(* CODESYS project Tc3_Physics.library
   TcLibraryId: Beckhoff Automation GmbH|Tc3_Physics|0.3.79.0
   Company: Beckhoff Automation GmbH
   DefaultNamespace: Tc3_Physics
   Version: 0.3.79.0
   Placeholder: Tc3_Physics
   Title: Tc3_Physics

Project tree, tasks and I/O mapping:
  Version/
    global variables Global_Version
  POUs/
    Spatial/
      Functions/
        function ConcatenateXY [ST]
        function Concatenate3D [ST]
        function ConcatenateC [ST]
        function ConcatenateABC [ST]
        function ConcatenateXYC [ST]
        function Concatenate6D [ST]
        function AddXY [ST]
        function SubtractXY [ST]
        function MultiplyXY [ST]
        function ScalarXY [ST]
        function Add3D [ST]
        function Subtract3D [ST]
        function Multiply3D [ST]
        function Scalar3D [ST]
        function Cross3D [ST]
        function AddABC [ST]
        function SubtractABC [ST]
        function MultiplyABC [ST]
        function AddXYC [ST]
        function SubtractXYC [ST]
        function MultiplyXYC [ST]
        function Add6D [ST]
        function Subtract6D [ST]
        function Multiply6D [ST]
        function ConvertToCartesian2D [ST]
      Positions/
        function block PositionXY [ST]: FB_init, FB_reinit, FB_exit, SetZero, SetValues, SetValuesXY, SetValuesRP, SetValuesXYReferenceId, GetRadius, GetPhi, Invert, ConcatenateWith, ShiftBy, ShiftByXY, x, y, ReferenceId
        function block Position3D [ST]: FB_init, FB_exit, SetZero, SetValues, SetValuesXYZ, SetValuesRPZ, SetValuesRTP, Invert, ConcatenateWith, ShiftBy, ShiftByXYZ, x, y, z
        function block Orientation2D [ST]: FB_init, FB_exit, SetAngle, SetZero, SetValues, GetDirectionX, GetDirectionY, Invert, ConcatenateWith, TurnByC, Transform, angle
        function block Orientation3D [ST]: FB_init, FB_exit, SetZero, SetValues, SetValuesABC, SetValuesACB, SetValuesBCA, SetValuesBAC, SetValuesCAB, SetValuesCBA, SetValuesABA, SetValuesACA, SetValuesBCB, SetValuesBAB, SetValuesCAC, SetValuesCBC, GetDirectionX, GetDirectionY, GetDirectionZ, Invert, ConcatenateWith, TurnBy, TurnByA, TurnByB, TurnByC, Transform, phi0, phi1, phi2, convention
        function block PositionXYC [ST]: FB_init, FB_reinit, FB_exit, SetZero, SetValues, SetValuesXY, SetValuesXYC, SetValuesXYCReferenceId, GetDirectionX, GetDirectionY, Invert, ConcatenateWith, StepByLocal, StepByLocalXY, ShiftBy, ShiftByXY, TurnByC, Transform, x, y, c, ReferenceId
        function block PositionSE3 [ST]: FB_init, FB_exit, SetZero, SetValues, SetValuesXYZ, SetValuesRPZ, SetValuesRTP, SetValuesABC, SetValuesACB, SetValuesBCA, SetValuesBAC, SetValuesCAB, SetValuesCBA, SetValuesABA, SetValuesACA, SetValuesBCB, SetValuesBAB, SetValuesCAC, SetValuesCBC, GetDirectionX, GetDirectionY, GetDirectionZ, Invert, ConcatenateWith, StepByLocal, StepByLocalXYZ, ShiftBy, ShiftByXYZ, TurnBy, TurnByA, TurnByB, TurnByC, Transform, x, y, z, phi0, phi1, phi2, Convention
      Tangents/
        function block TangentXY [ST]: FB_init, FB_exit, SetZero, SetValues, SetValuesXY, IsZero, GetLength, GetDirection, AddBy, AddByXY, SubtractBy, SubtractByXY, MultiplyBy, Normalize, x, y
        function block Tangent3D [ST]: FB_init, FB_exit, SetZero, SetValues, SetValuesXYZ, IsZero, GetLength, GetDirection, AddBy, AddByXYZ, SubtractBy, SubtractByXYZ, MultiplyBy, DivideBy, Normalize, x, y, z
        function block TangentABC [ST]: FB_init, FB_exit, SetZero, SetValues, SetValuesABC, IsZero, GetLength, AddBy, AddByABC, SubtractBy, SubtractByABC, MultiplyBy, a, b, c
        function block TangentXYC [ST]: FB_init, FB_exit, SetZero, SetValues, SetValuesXYC, IsZero, AddBy, AddByXYC, SubtractBy, SubtractByXYC, MultiplyBy, x, y, c
        function block Tangent6D [ST]: FB_init, FB_exit
      Setpoints/
        function block SetpointR1 [ST]: FB_init, FB_reinit, FB_exit, SetZero, SetValuesSVAJ, _s, v, a, j
        function block SetpointSE3 [ST]: FB_init, FB_exit, SetIdentity, SetValues, SetValuesXYZ, SetValuesCBA, GetDirectionX, GetDirectionY, GetDirectionZ, GetPosition_Cartesian, GetVelocity_Cartesian, GetAcceleration_Cartesian, GetJerk_Cartesian, ConcatenateWith, x, y, z, phi0, phi1, phi2, Convention
      Inertias/
        function block InertiaSE3 [ST]: FB_init, FB_exit, AddBy, SetValues_Point, SetValues_Sphere, SetValues_Cylinder, SetValues_Cuboid, Transform, Translate, mass, x, y, z, xx, yy, zz, xy, yz, zx
    _Internal/
      function block IPlcGeometry2D [ST]: FB_init, FB_exit
      function block IPlcGeometry3D [ST]: FB_init, FB_exit
      function block Geometry2D [ST]: FB_init, FB_exit, SetDisplacement, SetDisplacementXYC, SetDisplacementXY, SetDisplacementX, SetDisplacementY, SetDisplacementC, SetPosition, SetPositionXYC, SetPositionXY, SetPositionX, SetPositionY, SetPositionC, GetDisplacement, GetDisplacementX, GetDisplacementY, GetDisplacementC, GetLocalX, GetLocalY, GetPosition, GetPositionX, GetPositionY, GetPositionC, GetDirectionX, GetDirectionY, StepByLocal, StepByLocalXY, ShiftBy, ShiftByXY, TurnByC
      function block Geometry3D [ST]: FB_init, FB_exit, SetDisplacement, SetDisplacementXYZ, SetDisplacementX, SetDisplacementY, SetDisplacementZ, SetPosition, SetPositionXYZ, SetPositionX, SetPositionY, SetPositionZ, SetRotationABC, SetRotationACB, SetRotationBCA, SetRotationBAC, SetRotationCAB, SetRotationCBA, SetRotationABA, SetRotationACA, SetRotationBCB, SetRotationBAB, SetRotationCAC, SetRotationCBC, GetDisplacement, GetDisplacementX, GetDisplacementY, GetDisplacementZ, GetLocalX, GetLocalY, GetLocalZ, GetPosition, GetPositionX, GetPositionY, GetPositionZ, GetDirectionX, GetDirectionY, GetDirectionZ, StepByLocal, StepByLocalXYZ, ShiftBy, ShiftByXYZ, TurnBy, TurnByA, TurnByB, TurnByC, phi0, phi1, phi2, Convention
      function block IPlcPath2D [ST]: FB_init, FB_exit, CloseLoop, Clear, GetLength, IsClosedLoop, IsSelfColliding, GetArcLength_ClosestTo
      function block IPlcPath3D [ST]: FB_init, FB_exit, CloseLoop, Clear, GetLength, IsClosedLoop, IsSelfColliding, GetArcLength_ClosestTo
      function block IPlcDynamicConstraint [ST]: FB_init, FB_exit
    Shapes/
      Geometry2D/
        1D/
          function block Line2D [ST]: FB_init, FB_exit, DefineByPositions, DefineByDirection, SetDirection, GetDirection, GetPositionAt
          function block Segment2D [ST]: FB_init, FB_exit, SetStartPosition, SetStartPositionXY, SetEndPosition, SetEndPositionXY, Get_dX, Get_dY, GetLength, GetStartPosition, GetEndPosition, GetDirection, GetPositionAt
          function block Circle2D [ST]: FB_init, FB_exit, GetLength, GetPositionAt, radius
        2D/
          function block Disc2D [ST]: FB_init, FB_exit, GetArea, radius
          function block Rectangle2D [ST]: FB_init, FB_exit, SetDimensions, GetArea, width, height
        function block Container2D [ST]: FB_init, FB_exit, AddElement, RemoveElement, Clear, GetCount, GetBoundary
        function block Extrude2D [ST]: FB_init, FB_exit, ExtrudeAlong, IsValid
        Functions/
          function CheckCollision2D [ST]
          function GetDistance2D [ST]
          function GetLinkingLine2D [ST]
      Geometry3D/
        1D/
          function block Line3D [ST]: FB_init, FB_exit, DefineByPositions, DefineByDirection, SetDirection, GetDirection, GetPositionAt
          function block Segment3D [ST]: FB_init, FB_exit, SetStartPosition, SetStartPositionXYZ, SetEndPosition, SetEndPositionXYZ, Get_dX, Get_dY, Get_dZ, GetLength, GetStartPosition, GetEndPosition, GetDirection, GetPositionAt
          function block Circle3D [ST]: FB_init, FB_exit, SetNormal, GetLength, GetNormal, GetPositionAt, radius
        2D/
          function block Plane3D [ST]: FB_init, FB_exit, SetNormal, GetNormal
          function block Disc3D [ST]: FB_init, FB_exit, SetNormal, GetNormal, GetArea, radius
          function block Rectangle3D [ST]: FB_init, FB_exit, SetDimensions, GetArea, width, height
        3D/
          function block Sphere3D [ST]: FB_init, FB_exit, GetVolume, radius
          function block Cuboid3D [ST]: FB_init, FB_exit, SetDimensions, GetVolume, length, width, height
          function block Cylinder3D [ST]: FB_init, FB_exit, SetDimensions, GetVolume, radius, height
        function block Container3D [ST]: FB_init, FB_exit, AddElement, RemoveElement, Clear, GetCount
        function block Extrude3D [ST]: FB_init, FB_exit, DefineByPath
        Functions/
          function CheckCollision3D [ST]
          function GetDistance3D [ST]
          function GetLinkingLine3D [ST]
          function CreateIntersection2D [ST]
    Paths/
      Components/
        function block PathXY [ST]: FB_init, FB_exit, AppendPosition, AppendPositionXY, AppendLine, AppendCircle, GetStartPosition, GetEndPosition, GetPositionAt, GetStateAt
        function block PathXYC [ST]: FB_init, FB_exit, AppendPosition, AppendPositionXYC, AppendLine, AppendCircle, EndAtPath, StartFromPath, CloseLoop, Clear, GetStartPosition, GetEndPosition, GetPositionAt, GetStateAt
        function block PathXYZ [ST]: FB_init, FB_exit, AppendPosition, AppendPositionXYZ, AppendLine, AppendLineXYZ, AppendCircle, AppendPositionTangent, GetStartPosition, GetEndPosition, GetPositionAt, GetStateAt
    Dynamics/
      function block DynamicConstraint_Container [ST]: FB_init, FB_exit, Clear, AddConstraint, AddConstraintByReference, Count
      function block DynamicConstraint_CartesianXY [ST]: FB_init, FB_exit, SetValuesVAJ, V, A, J
      function block DynamicConstraint_CartesianXYZ [ST]: FB_init, FB_exit, SetValuesVAJ, V, A, J
      function block DynamicConstraint_Path [ST]: FB_init, FB_exit
      function block DynamicConstraint_PathXY [ST]: FB_init, FB_exit, SetValuesVADJ, V, A, D, J
      function block DynamicConstraint_PathXYZ [ST]: FB_init, FB_exit, SetValuesVADJ, V, A, D, J
      function block DynamicConstraint_Coordinates [ST]: FB_init, FB_exit, AddLimit, SetLimit, RemoveLimit, Clear, GetV, GetA, GetD, GetJ, Count
      function block DynamicProfile_7phase [ST]: FB_init, FB_exit, SetDynamicLimits, CalculateProfile, GetValues, GetDuration
      function block DynamicProfile_3phase [ST]: FB_init, FB_exit, SetDynamicLimits, CalculateProfile, GetValues, GetDuration
    Coordinates/
      function GetMcsCoordinateType [ST]
      function GetUninterpretedCoordinateType [ST]
  DUTs/
    Enumerations/
      data type E_RotationCoordinates
      data type E_CoordCategory
      data type E_McsCoordType
    data type CoordinateType
  GVLs/
    global variables GVL
*)

// DUTs/CoordinateType

(* Coordinate type. Use provided constants such as Coord_Mcs_X or factory functions such as GetMcsCoordinateType for creation. *)
	{attribute 'TcIecLibraryType'}
TYPE CoordinateType : 
	STRUCT
		(* Reserved. *)
		{attribute 'hide'}
		_reserved0 : ULINT := 0;
	END_STRUCT
END_TYPE

// DUTs/Enumerations/E_RotationCoordinates

(* Enumeration of rotation conventions. 
			    The order of letters defines the order of rotation around local axes.
			    This also defines order in which user should program rotation values. *)
	{attribute 'TcIecLibraryType'}
{attribute 'qualified_only'}
{attribute 'strict'}
TYPE E_RotationCoordinates : (
	ABC:=0, 	(* ABC *)
	ACB:=1, 	(* ACB *)
	BCA:=2, 	(* BCA *)
	BAC:=3, 	(* BAC *)
	CAB:=4, 	(* CAB *)
	CBA:=5, 	(* CBA *)
	ABA:=6, 	(* ABA *)
	ACA:=7, 	(* ACA *)
	BCB:=8, 	(* BCB *)
	BAB:=9, 	(* BAB *)
	CAC:=10, 	(* CAC *)
	CBC:=11	(* CBC *)
) UDINT;
END_TYPE

// DUTs/Enumerations/E_CoordCategory

(* Enumeration coordinate categories. *)
	{attribute 'TcIecLibraryType'}
{attribute 'qualified_only'}
{attribute 'strict'}
TYPE E_CoordCategory : (
	Invalid:=16#0, 	(* Invalid *)
	MCS:=16#1, 	(* MCS *)
	ACS:=16#2, 	(* ACS *)
	Uninterpreted:=16#3	(* Uninterpreted *)
) UDINT;
END_TYPE

// DUTs/Enumerations/E_McsCoordType

(* Enumeration of MCS coordinate types. *)
	{attribute 'TcIecLibraryType'}
{attribute 'qualified_only'}
{attribute 'strict'}
TYPE E_McsCoordType : (
	Invalid:=16#0, 	(* Invalid *)
	X:=16#11, 	(* X *)
	Y:=16#21, 	(* Y *)
	Z:=16#31, 	(* Z *)
	A1:=16#41, 	(* A1 *)
	A2:=16#42, 	(* A2 *)
	A3:=16#43, 	(* A3 *)
	B1:=16#51, 	(* B1 *)
	B2:=16#52, 	(* B2 *)
	B3:=16#53, 	(* B3 *)
	C1:=16#61, 	(* C1 *)
	C2:=16#62, 	(* C2 *)
	C3:=16#63	(* C3 *)
) UDINT;
END_TYPE

// Version/Global_Version
{attribute 'TcGenerated'}
// This function has been automatically generated from the project information.
VAR_GLOBAL CONSTANT
	{attribute 'const_non_replaced'}
	{attribute 'linkalways'}
	stLibVersion_Tc3_Physics : ST_LibVersion := (iMajor := 0, iMinor := 3, iBuild := 79, iRevision := 0, sVersion := '0.3.79.0');
	{attribute 'const_non_replaced'}
	{attribute 'linkalways'}
	sLibraryId_Tc3_Physics : String := 'Beckhoff Automation GmbH|Tc3_Physics|0.3.79.0';
END_VAR

// GVLs/GVL

VAR_GLOBAL CONSTANT
		Coord_Mcs_X	:	CoordinateType := GetMcsCoordinateType(E_McsCoordType.X);
		Coord_Mcs_Y	:	CoordinateType := GetMcsCoordinateType(E_McsCoordType.Y);
		Coord_Mcs_Z	:	CoordinateType := GetMcsCoordinateType(E_McsCoordType.Z);
		Coord_Mcs_A1	:	CoordinateType := GetMcsCoordinateType(E_McsCoordType.A1);
		Coord_Mcs_A2	:	CoordinateType := GetMcsCoordinateType(E_McsCoordType.A2);
		Coord_Mcs_A3	:	CoordinateType := GetMcsCoordinateType(E_McsCoordType.A3);
		Coord_Mcs_B1	:	CoordinateType := GetMcsCoordinateType(E_McsCoordType.B1);
		Coord_Mcs_B2	:	CoordinateType := GetMcsCoordinateType(E_McsCoordType.B2);
		Coord_Mcs_B3	:	CoordinateType := GetMcsCoordinateType(E_McsCoordType.B3);
		Coord_Mcs_C1	:	CoordinateType := GetMcsCoordinateType(E_McsCoordType.C1);
		Coord_Mcs_C2	:	CoordinateType := GetMcsCoordinateType(E_McsCoordType.C2);
		Coord_Mcs_C3	:	CoordinateType := GetMcsCoordinateType(E_McsCoordType.C3);
		Coord_Uninterpreted1	:	CoordinateType := GetUninterpretedCoordinateType(1);
		Coord_Uninterpreted2	:	CoordinateType := GetUninterpretedCoordinateType(2);
		Coord_Uninterpreted3	:	CoordinateType := GetUninterpretedCoordinateType(3);
		Coord_Uninterpreted4	:	CoordinateType := GetUninterpretedCoordinateType(4);
		Coord_Uninterpreted5	:	CoordinateType := GetUninterpretedCoordinateType(5);
		Coord_Uninterpreted6	:	CoordinateType := GetUninterpretedCoordinateType(6);
		Coord_Uninterpreted7	:	CoordinateType := GetUninterpretedCoordinateType(7);
		Coord_Uninterpreted8	:	CoordinateType := GetUninterpretedCoordinateType(8);
	END_VAR

// POUs/_Internal/IPlcGeometry2D

	{attribute 'c++_compatible'}
	{attribute 'external_name' := 'IPlcGeometry2D_GUID_0554E5C0_4687_0E31_67FE_D976C958432A'}
	{attribute 'TcIecLibraryType'}
	{attribute 'no_explicit_call' :='do not call this POU directly'}
	{attribute 'no_assign_warning'}
	(* Internal representation of an object in the planar space. *)
	FUNCTION_BLOCK IPlcGeometry2D
	VAR
		(* x-coordinate of the instance. *)
		px : LREAL;
		(* y-coordinate of the instance. *)
		py : LREAL;
		(* c-rotation of the instance given in degrees [Â°]. *)
		pc : LREAL;
		 {attribute 'hide'}
		_reserved1 : ARRAY [1..24] OF USINT;
	END_VAR
	VAR_OUTPUT
		(* ErrorCode for last method execution *)
		nErrorId : UDINT;
		(* Error during last method execution *)
		bError : BOOL;
	END_VAR
	VAR
		 {attribute 'hide'}
		_reserved2 : ARRAY [1..35] OF USINT;
	END_VAR


	(* Internal method *)
	{attribute 'hide'}
	METHOD FB_init : BOOL
	VAR_INPUT
		(*  if TRUE, the retain variables are initialized (warm start / cold start) *)
		bInitRetains : BOOL;
		(*  if TRUE, the instance afterwards gets moved into the copy code (online change) *)
		bInCopyCode : BOOL;
	END_VAR
END_METHOD


	(* Internal method *)
	{attribute 'hide'}
	METHOD FB_exit : BOOL
	VAR_INPUT
		(*  if TRUE, the exit method is called for exiting an instance that is copied afterwards (online change). *)
		bInCopyCode : BOOL;
	END_VAR
END_METHOD

END_FUNCTION_BLOCK

// POUs/_Internal/IPlcGeometry3D

	{attribute 'c++_compatible'}
	{attribute 'external_name' := 'IPlcGeometry3D_GUID_353920C5_B103_0C39_7785_16CAA850CA31'}
	{attribute 'TcIecLibraryType'}
	{attribute 'no_explicit_call' :='do not call this POU directly'}
	{attribute 'no_assign'}
	(* Internal representation of an object in the 3D space. *)
	FUNCTION_BLOCK IPlcGeometry3D
	VAR
		(* x-coordinate of the instance. *)
		px : LREAL;
		(* y-coordinate of the instance. *)
		py : LREAL;
		(* z-coordinate of the instance. *)
		pz : LREAL;
		 {attribute 'hide'}
		_reserved1 : ARRAY [1..40] OF USINT;
	END_VAR
	VAR_OUTPUT
		(* ErrorCode for last method execution *)
		nErrorId : UDINT;
		(* Error during last method execution *)
		bError : BOOL;
	END_VAR
	VAR
		 {attribute 'hide'}
		_reserved2 : ARRAY [1..43] OF USINT;
	END_VAR


	(* Internal method *)
	{attribute 'hide'}
	METHOD FB_init : BOOL
	VAR_INPUT
		(*  if TRUE, the retain variables are initialized (warm start / cold start) *)
		bInitRetains : BOOL;
		(*  if TRUE, the instance afterwards gets moved into the copy code (online change) *)
		bInCopyCode : BOOL;
	END_VAR
END_METHOD


	(* Internal method *)
	{attribute 'hide'}
	METHOD FB_exit : BOOL
	VAR_INPUT
		(*  if TRUE, the exit method is called for exiting an instance that is copied afterwards (online change). *)
		bInCopyCode : BOOL;
	END_VAR
END_METHOD

END_FUNCTION_BLOCK

// POUs/_Internal/Geometry2D

	{attribute 'c++_compatible'}
	{attribute 'external_name' := 'Geometry2D_GUID_EA1925AE_2507_0F27_40AC_5A565B8F6BBE'}
	{attribute 'TcIecLibraryType'}
	{attribute 'no_explicit_call' :='do not call this POU directly'}
	{attribute 'no_assign'}
	(* Base class for all 2D simple geometries (all dimensions, line etc.) *)
	FUNCTION_BLOCK Geometry2D EXTENDS IPlcGeometry2D


	(* Internal method *)
	METHOD FB_init : BOOL
	VAR_INPUT
		(*  if TRUE, the retain variables are initialized (warm start / cold start) *)
		bInitRetains : BOOL;
		(*  if TRUE, the instance afterwards gets moved into the copy code (online change) *)
		bInCopyCode : BOOL;
	END_VAR
END_METHOD


	(* Internal method *)
	{attribute 'hide'}
	METHOD FB_exit : BOOL
	VAR_INPUT
		(*  if TRUE, the exit method is called for exiting an instance that is copied afterwards (online change). *)
		bInCopyCode : BOOL;
	END_VAR
END_METHOD


	(* Set the position of this geometry in respect to the reference frame. *)
	METHOD SetDisplacement
	VAR_IN_OUT
		(* The displacement to set. *)
 {attribute 'GUID' := '54EDED35-5A53-0913-4680-EA5D332AAA4F'}
				displacement : PositionXYC;
	END_VAR
END_METHOD


	(* Set the position of this geometry in respect to the reference frame. *)
	METHOD SetDisplacementXYC
	VAR_INPUT
		(* x-component of the position. *)
		x : LREAL;
		(* y-component of the position. *)
		y : LREAL;
		(* c-component of the position given in degrees [Â°]. *)
		c : LREAL;
	END_VAR
END_METHOD


	(* Set the position of this geometry in respect to the reference frame. *)
	METHOD SetDisplacementXY
	VAR_INPUT
		(* x-component of the position. *)
		x : LREAL;
		(* y-component of the position. *)
		y : LREAL;
	END_VAR
END_METHOD


	(* Set the local x-coordinate of this geometry. *)
	METHOD SetDisplacementX
	VAR_INPUT
		(* Global x-component of the position. *)
		x : LREAL;
	END_VAR
END_METHOD


	(* Set the local y-coordinate of this geometry. *)
	METHOD SetDisplacementY
	VAR_INPUT
		(* Global y-component of the position. *)
		y : LREAL;
	END_VAR
END_METHOD


	(* Set the local c-component of this geometry. *)
	METHOD SetDisplacementC
	VAR_INPUT
		(* c-orientation given in degrees [Â°]. *)
		c : LREAL;
	END_VAR
END_METHOD


	(* Set the position of this geometry in respect to the WCS. *)
	METHOD SetPosition
	VAR_IN_OUT
		(* The position to set. *)
 {attribute 'GUID' := '54EDED35-5A53-0913-4680-EA5D332AAA4F'}
				position : PositionXYC;
	END_VAR
END_METHOD


	(* Set the position of this geometry in respect to the WCS. *)
	METHOD SetPositionXYC
	VAR_INPUT
		(* x-component of the position. *)
		x : LREAL;
		(* y-component of the position. *)
		y : LREAL;
		(* c-component of the position given in degrees [Â°]. *)
		c : LREAL;
	END_VAR
END_METHOD


	(* Set the position of this geometry in respect to the WCS. *)
	METHOD SetPositionXY
	VAR_INPUT
		(* x-component of the position. *)
		x : LREAL;
		(* y-component of the position. *)
		y : LREAL;
	END_VAR
END_METHOD


	(* Set the global x-coordinate of this geometry. *)
	METHOD SetPositionX
	VAR_INPUT
		(* Global x-component of the position. *)
		x : LREAL;
	END_VAR
END_METHOD


	(* Set the global y-coordinate of this geometry. *)
	METHOD SetPositionY
	VAR_INPUT
		(* Global y-component of the position. *)
		y : LREAL;
	END_VAR
END_METHOD


	(* Set the global c-component of this geometry. *)
	METHOD SetPositionC
	VAR_INPUT
		(* c-orientation given in degrees [Â°]. *)
		c : LREAL;
	END_VAR
END_METHOD


	(* Get the position of this geometry in respect to the reference frame. *)
	METHOD GetDisplacement
	VAR_IN_OUT
		(* The current position of the geometry. *)
 {attribute 'GUID' := '54EDED35-5A53-0913-4680-EA5D332AAA4F'}
				displacement : PositionXYC;
	END_VAR
END_METHOD


	(* Get the local x-component of this geometry. *)
	METHOD GetDisplacementX : LREAL
END_METHOD


	(* Get the local y-component of this geometry. *)
	METHOD GetDisplacementY : LREAL
END_METHOD


	(* Get the local c-orientation of this geometry. *)
	METHOD GetDisplacementC : LREAL
END_METHOD


	(* Get the direction of the local x-axis. *)
	METHOD GetLocalX
	VAR_IN_OUT
		(* The local x-direction of this geometry. *)
 {attribute 'GUID' := '619D5D7D-53EC-0B73-54D5-FB9C43AFDE82'}
				localX : TangentXY;
	END_VAR
END_METHOD


	(* Get the direction of the local y-axis. *)
	METHOD GetLocalY
	VAR_IN_OUT
		(* The local y-direction of this geometry. *)
 {attribute 'GUID' := '619D5D7D-53EC-0B73-54D5-FB9C43AFDE82'}
				localY : TangentXY;
	END_VAR
END_METHOD


	(* Get the position of this geometry. *)
	METHOD GetPosition
	VAR_IN_OUT
		(* The current position of the geometry. *)
 {attribute 'GUID' := '54EDED35-5A53-0913-4680-EA5D332AAA4F'}
				position : PositionXYC;
	END_VAR
END_METHOD


	(* Get the global x-component of this geometry. *)
	METHOD GetPositionX : LREAL
END_METHOD


	(* Get the global y-component of this geometry. *)
	METHOD GetPositionY : LREAL
END_METHOD


	(* Get the global c-orientation of this geometry. *)
	METHOD GetPositionC : LREAL
END_METHOD


	(* Get the direction of the local x-axis. *)
	METHOD GetDirectionX
	VAR_IN_OUT
		(* The global x-direction of this geometry. *)
 {attribute 'GUID' := '619D5D7D-53EC-0B73-54D5-FB9C43AFDE82'}
				directionX : TangentXY;
	END_VAR
END_METHOD


	(* Get the direction of the local y-axis. *)
	METHOD GetDirectionY
	VAR_IN_OUT
		(* The global y-direction of this geometry. *)
 {attribute 'GUID' := '619D5D7D-53EC-0B73-54D5-FB9C43AFDE82'}
				directionY : TangentXY;
	END_VAR
END_METHOD


	(* Displace the components of this position. The shift is applied within the local coordinate frame. *)
	METHOD StepByLocal
	VAR_IN_OUT
		(* The displacement to shift by. *)
 {attribute 'GUID' := 'E037A91B-C1D8-04E4-4DB7-2726DA6E0D41'}
				shift : TangentXYC;
	END_VAR
END_METHOD


	(* Apply a local step in respect to the local coordinate frame without changing the orientation. *)
	METHOD StepByLocalXY
	VAR_INPUT
		(* The displacement within the local x-direction. *)
		dx : LREAL;
		(* The displacement within the local y-direction. *)
		dy : LREAL;
	END_VAR
END_METHOD


	(* Displace the components of this position. *)
	METHOD ShiftBy
	VAR_IN_OUT
		(* Shift vector to displace by. *)
 {attribute 'GUID' := '619D5D7D-53EC-0B73-54D5-FB9C43AFDE82'}
				shift : TangentXY;
	END_VAR
END_METHOD


	(* Displace the components of this position. *)
	METHOD ShiftByXY
	VAR_INPUT
		(* Shift of the x-component of this position. *)
		dx : LREAL;
		(* Shift of the y-component of this position. *)
		dy : LREAL;
	END_VAR
END_METHOD


	(* Rotate the attached orientation without changing the Cartesian coodinates. *)
	METHOD TurnByC
	VAR_INPUT
		(* Angular displacement given in degrees [Â°]. *)
		dc : LREAL;
	END_VAR
END_METHOD

END_FUNCTION_BLOCK

// POUs/Spatial/Positions/PositionXYC

	{attribute 'c++_compatible'}
	{attribute 'external_name' := 'PositionXYC_GUID_54EDED35_5A53_0913_4680_EA5D332AAA4F'}
	{attribute 'TcIecLibraryType'}
	{attribute 'no_explicit_call' :='do not call this POU directly'}
	{attribute 'no_assign_warning'}
	(* A position in the xy-plane with an in-plane direction c. *)
	FUNCTION_BLOCK PositionXYC EXTENDS IPlcGeometry2D


	(* Internal method *)
	{attribute 'hide'}
	METHOD FB_init : BOOL
	VAR_INPUT
		(*  if TRUE, the retain variables are initialized (warm start / cold start) *)
		bInitRetains : BOOL;
		(*  if TRUE, the instance afterwards gets moved into the copy code (online change) *)
		bInCopyCode : BOOL;
	END_VAR
END_METHOD


	(* Internal method *)
	{attribute 'hide'}
	METHOD FB_reinit : BOOL
END_METHOD


	(* Internal method *)
	{attribute 'hide'}
	METHOD FB_exit : BOOL
	VAR_INPUT
		(*  if TRUE, the exit method is called for exiting an instance that is copied afterwards (online change). *)
		bInCopyCode : BOOL;
	END_VAR
END_METHOD


	(* Set the components of this vector to '0.0'. *)
	METHOD SetZero
END_METHOD


	(* Set the components of this position. *)
	METHOD SetValues
	VAR_IN_OUT
		(* The values to set. *)
 {attribute 'GUID' := '54EDED35-5A53-0913-4680-EA5D332AAA4F'}
				positionXYC : PositionXYC;
	END_VAR
END_METHOD


	(* Set the spatial components of this position. *)
	METHOD SetValuesXY
	VAR_INPUT
		(* x-component of the position. *)
		x : LREAL;
		(* y-component of the position. *)
		y : LREAL;
	END_VAR
END_METHOD


	(* Set the components of this position. *)
	METHOD SetValuesXYC
	VAR_INPUT
		(* x-component of the position. *)
		x : LREAL;
		(* y-component of the position. *)
		y : LREAL;
		(* c-component of the position scaled in degrees [Â°]. *)
		c : LREAL;
	END_VAR
END_METHOD


	(* Set the components of this position. *)
	METHOD SetValuesXYCReferenceId
	VAR_INPUT
		(* x-component of the position. *)
		x : LREAL;
		(* y-component of the position. *)
		y : LREAL;
		(* c-component of the position scaled in degrees [Â°]. *)
		c : LREAL;
		(* reference id of the position. *)
 {attribute 'GUID' := '18071995-0000-0000-0000-00000000000F'}
				ReferenceId : OTCID;
	END_VAR
END_METHOD


	(* Get the direction of the local x-axis. *)
	METHOD GetDirectionX
	VAR_IN_OUT
		(* The local x-direction of this position. *)
 {attribute 'GUID' := '619D5D7D-53EC-0B73-54D5-FB9C43AFDE82'}
				localX : TangentXY;
	END_VAR
END_METHOD


	(* Get the direction of the local y-axis. *)
	METHOD GetDirectionY
	VAR_IN_OUT
		(* The local y-direction of this position. *)
 {attribute 'GUID' := '619D5D7D-53EC-0B73-54D5-FB9C43AFDE82'}
				localY : TangentXY;
	END_VAR
END_METHOD


	(* Invert this position. *)
	METHOD Invert
END_METHOD


	(* Multiply this position by a 2nd from the right. *)
	METHOD ConcatenateWith
	VAR_IN_OUT
		(* The position to concatenate with. *)
 {attribute 'GUID' := '54EDED35-5A53-0913-4680-EA5D332AAA4F'}
				position : PositionXYC;
	END_VAR
END_METHOD


	(* Displace the components of this position. The shift is applied within the local coordinate frame. *)
	METHOD StepByLocal
	VAR_IN_OUT
		(* The displacement to shift by. *)
 {attribute 'GUID' := 'E037A91B-C1D8-04E4-4DB7-2726DA6E0D41'}
				shift : TangentXYC;
	END_VAR
END_METHOD


	(* Apply a local step in respect to the local coordinate frame without changing the orientation. *)
	METHOD StepByLocalXY
	VAR_INPUT
		(* The displacement within the local x-direction. *)
		dx : LREAL;
		(* The displacement within the local y-direction. *)
		dy : LREAL;
	END_VAR
END_METHOD


	(* Displace the components of this position. *)
	METHOD ShiftBy
	VAR_IN_OUT
		(* Shift vector to displace by. *)
 {attribute 'GUID' := '619D5D7D-53EC-0B73-54D5-FB9C43AFDE82'}
				shift : TangentXY;
	END_VAR
END_METHOD


	(* Displace the components of this position. *)
	METHOD ShiftByXY
	VAR_INPUT
		(* Shift of the x-component of this position. *)
		dx : LREAL;
		(* Shift of the y-component of this position. *)
		dy : LREAL;
	END_VAR
END_METHOD


	(* Rotate the attached orientation without changing the Cartesian coodinates. *)
	METHOD TurnByC
	VAR_INPUT
		(* Angular displacement given in degrees [Â°]. *)
		dc : LREAL;
	END_VAR
END_METHOD


	(* Place a PositionXY into the coordinate system referenced by this position. *)
	METHOD Transform
	VAR_IN_OUT
		(* Position to transform. *)
 {attribute 'GUID' := 'D1D75488-37B1-0155-53AF-A9A9BDBB4FFD'}
				positionXY : PositionXY;
	END_VAR
END_METHOD


	PROPERTY x : LREAL
GET
END_GET
SET
END_SET
END_PROPERTY


	PROPERTY y : LREAL
GET
END_GET
SET
END_SET
END_PROPERTY


	PROPERTY c : LREAL
GET
END_GET
SET
END_SET
END_PROPERTY


{attribute 'monitoring' := 'call'}
	PROPERTY ReferenceId : OTCID
GET
END_GET
SET
END_SET
END_PROPERTY

END_FUNCTION_BLOCK

// POUs/Spatial/Tangents/TangentXY

	{attribute 'c++_compatible'}
	{attribute 'external_name' := 'TangentXY_GUID_619D5D7D_53EC_0B73_54D5_FB9C43AFDE82'}
	{attribute 'TcIecLibraryType'}
	{attribute 'no_explicit_call' :='do not call this POU directly'}
	{attribute 'no_assign'}
	(* A Cartesian direction vector to describe a displacement of velocity in the 2D-Cartesian space. *)
	FUNCTION_BLOCK TangentXY
	VAR
		(* x-component of the tangent. *)
		dx : LREAL;
		(* y-component of the tangent. *)
		dy : LREAL;
		 {attribute 'hide'}
		_reserved1 : ARRAY [1..72] OF USINT;
	END_VAR


	(* Internal method *)
	{attribute 'hide'}
	METHOD FB_init : BOOL
	VAR_INPUT
		(*  if TRUE, the retain variables are initialized (warm start / cold start) *)
		bInitRetains : BOOL;
		(*  if TRUE, the instance afterwards gets moved into the copy code (online change) *)
		bInCopyCode : BOOL;
	END_VAR
END_METHOD


	(* Internal method *)
	{attribute 'hide'}
	METHOD FB_exit : BOOL
	VAR_INPUT
		(*  if TRUE, the exit method is called for exiting an instance that is copied afterwards (online change). *)
		bInCopyCode : BOOL;
	END_VAR
END_METHOD


	(* Set the components of this tangent to '0.0'. *)
	METHOD SetZero
END_METHOD


	(* Set the components of this tangent. *)
	METHOD SetValues
	VAR_IN_OUT
		(* The tangent values to set. *)
 {attribute 'GUID' := '619D5D7D-53EC-0B73-54D5-FB9C43AFDE82'}
				tangentXY : TangentXY;
	END_VAR
END_METHOD


	(* Set the components of this tangent. *)
	METHOD SetValuesXY
	VAR_INPUT
		(* x-component of the tangent. *)
		x : LREAL;
		(* y-component of the tangent. *)
		y : LREAL;
	END_VAR
END_METHOD


	(* Check if all components of this tangent are within a tolerance from zero. *)
	METHOD IsZero : BOOL
	VAR_INPUT
		(* The tolerance threshold for each of the components. *)
		tolerance : LREAL;
	END_VAR
END_METHOD


	(* Get the Euclidean length of this tangent vector. *)
	METHOD GetLength : LREAL
END_METHOD


	(* Get the normalized direction to this tangent vector. *)
	METHOD GetDirection
	VAR_IN_OUT
		(* The normalized direction vector. *)
 {attribute 'GUID' := '619D5D7D-53EC-0B73-54D5-FB9C43AFDE82'}
				direction : TangentXY;
	END_VAR
END_METHOD


	(* Add a 2nd tangent vector to this one. *)
	METHOD AddBy
	VAR_IN_OUT
		(* The tangent vector to add. *)
 {attribute 'GUID' := '619D5D7D-53EC-0B73-54D5-FB9C43AFDE82'}
				shift : TangentXY;
	END_VAR
END_METHOD


	(* Add values to each of the components of this tangent vector. *)
	METHOD AddByXY
	VAR_INPUT
		(* Value to add to the x-component. *)
		dx : LREAL;
		(* Value to add to the y-component. *)
		dy : LREAL;
	END_VAR
END_METHOD


	(* Subtract a 2nd tangent vector from this one. *)
	METHOD SubtractBy
	VAR_IN_OUT
		(* The tangent vector to subtract. *)
 {attribute 'GUID' := '619D5D7D-53EC-0B73-54D5-FB9C43AFDE82'}
				shift : TangentXY;
	END_VAR
END_METHOD


	(* Subtract values from each of the components of this tangent vector. *)
	METHOD SubtractByXY
	VAR_INPUT
		(* Value to subtract from the x-component. *)
		dx : LREAL;
		(* Value to subtract from the y-component. *)
		dy : LREAL;
	END_VAR
END_METHOD


	(* Multiply the components of this tangent vector by a number. *)
	METHOD MultiplyBy
	VAR_INPUT
		(* The number to scale this tangent by. *)
		scale : LREAL;
	END_VAR
END_METHOD


	(* Normalize this tangent. *)
	METHOD Normalize
END_METHOD


	PROPERTY x : LREAL
GET
END_GET
SET
END_SET
END_PROPERTY


	PROPERTY y : LREAL
GET
END_GET
SET
END_SET
END_PROPERTY

END_FUNCTION_BLOCK

// POUs/Spatial/Tangents/TangentXYC

	{attribute 'c++_compatible'}
	{attribute 'external_name' := 'TangentXYC_GUID_E037A91B_C1D8_04E4_4DB7_2726DA6E0D41'}
	{attribute 'TcIecLibraryType'}
	{attribute 'no_explicit_call' :='do not call this POU directly'}
	{attribute 'no_assign'}
	(* An Euclidean direction to describe
				  a displacement or velocity in the local 2D-Cartesian space
				  with an additional angular displacement information. *)
	FUNCTION_BLOCK TangentXYC
	VAR
		(* x-component of the tangent *)
		dx : LREAL;
		(* y-component of the tangent *)
		dy : LREAL;
		(* c-component of the tangent in degree *)
		dc : LREAL;
		 {attribute 'hide'}
		_reserved1 : ARRAY [1..64] OF USINT;
	END_VAR


	(* Internal method *)
	{attribute 'hide'}
	METHOD FB_init : BOOL
	VAR_INPUT
		(*  if TRUE, the retain variables are initialized (warm start / cold start) *)
		bInitRetains : BOOL;
		(*  if TRUE, the instance afterwards gets moved into the copy code (online change) *)
		bInCopyCode : BOOL;
	END_VAR
END_METHOD


	(* Internal method *)
	{attribute 'hide'}
	METHOD FB_exit : BOOL
	VAR_INPUT
		(*  if TRUE, the exit method is called for exiting an instance that is copied afterwards (online change). *)
		bInCopyCode : BOOL;
	END_VAR
END_METHOD


	(* Set the components of this tangent to '0.0'. *)
	METHOD SetZero
END_METHOD


	(* Set the components of this tangent. *)
	METHOD SetValues
	VAR_IN_OUT
		(* The tangent values to set. *)
 {attribute 'GUID' := 'E037A91B-C1D8-04E4-4DB7-2726DA6E0D41'}
				tangentXYC : TangentXYC;
	END_VAR
END_METHOD


	(* Set the components of this tangent. *)
	METHOD SetValuesXYC
	VAR_INPUT
		(* x-component of the tangent. *)
		x : LREAL;
		(* y-component of the tangent. *)
		y : LREAL;
		(* c-component of the tangent in degrees [Â°]. *)
		c : LREAL;
	END_VAR
END_METHOD


	(* Check if all components of this tangent are within a tolerance from zero. *)
	METHOD IsZero : BOOL
	VAR_INPUT
		(* The tolerance threshold for each of the components. *)
		tolerance : LREAL;
	END_VAR
END_METHOD


	(* Add a 2nd tangent vector to this one. *)
	METHOD AddBy
	VAR_IN_OUT
		(* The tangent vector to add. *)
 {attribute 'GUID' := 'E037A91B-C1D8-04E4-4DB7-2726DA6E0D41'}
				shift : TangentXYC;
	END_VAR
END_METHOD


	(* Add values to each of the components of this tangent vector. *)
	METHOD AddByXYC
	VAR_INPUT
		(* Value to add to the x-component. *)
		dx : LREAL;
		(* Value to add to the y-component. *)
		dy : LREAL;
		(* Value to add to the c-component in degrees [Â°]. *)
		dc : LREAL;
	END_VAR
END_METHOD


	(* Subtract a 2nd tangent vector from this one. *)
	METHOD SubtractBy
	VAR_IN_OUT
		(* The tangent vector to subtract. *)
 {attribute 'GUID' := 'E037A91B-C1D8-04E4-4DB7-2726DA6E0D41'}
				shift : TangentXYC;
	END_VAR
END_METHOD


	(* Subtract values from each of the components of this tangent vector. *)
	METHOD SubtractByXYC
	VAR_INPUT
		(* Value to subtract from the x-component. *)
		dx : LREAL;
		(* Value to subtract from the y-component. *)
		dy : LREAL;
		(* Value to subtract from the c-component in degrees [Â°]. *)
		dc : LREAL;
	END_VAR
END_METHOD


	(* Multiply the components of this tangent vector by a number. *)
	METHOD MultiplyBy
	VAR_INPUT
		(* The number to scale this tangent by. *)
		scale : LREAL;
	END_VAR
END_METHOD


	PROPERTY x : LREAL
GET
END_GET
SET
END_SET
END_PROPERTY


	PROPERTY y : LREAL
GET
END_GET
SET
END_SET
END_PROPERTY


	PROPERTY c : LREAL
GET
END_GET
SET
END_SET
END_PROPERTY

END_FUNCTION_BLOCK

// POUs/Spatial/Positions/PositionXY

	{attribute 'c++_compatible'}
	{attribute 'external_name' := 'PositionXY_GUID_D1D75488_37B1_0155_53AF_A9A9BDBB4FFD'}
	{attribute 'TcIecLibraryType'}
	{attribute 'no_explicit_call' :='do not call this POU directly'}
	{attribute 'no_assign_warning'}
	(* Position in the 2D Cartesian space. *)
	FUNCTION_BLOCK PositionXY EXTENDS IPlcGeometry2D


	(* Internal method *)
	{attribute 'hide'}
	METHOD FB_init : BOOL
	VAR_INPUT
		(*  if TRUE, the retain variables are initialized (warm start / cold start) *)
		bInitRetains : BOOL;
		(*  if TRUE, the instance afterwards gets moved into the copy code (online change) *)
		bInCopyCode : BOOL;
	END_VAR
END_METHOD


	(* Internal method *)
	{attribute 'hide'}
	METHOD FB_reinit : BOOL
END_METHOD


	(* Internal method *)
	{attribute 'hide'}
	METHOD FB_exit : BOOL
	VAR_INPUT
		(*  if TRUE, the exit method is called for exiting an instance that is copied afterwards (online change). *)
		bInCopyCode : BOOL;
	END_VAR
END_METHOD


	(* Set the coordinates of this position to '0.0'. *)
	METHOD SetZero
END_METHOD


	(* Set the coordinates of this position. *)
	METHOD SetValues
	VAR_IN_OUT
		(* The coordinate values to set. *)
 {attribute 'GUID' := 'D1D75488-37B1-0155-53AF-A9A9BDBB4FFD'}
				positionXY : PositionXY;
	END_VAR
END_METHOD


	(* Set the xy-coordinates of this position. *)
	METHOD SetValuesXY
	VAR_INPUT
		(* x-component of the position. *)
		x : LREAL;
		(* y-component of the position. *)
		y : LREAL;
	END_VAR
END_METHOD


	(* Set the components of this position in polar coordinates. *)
	METHOD SetValuesRP
	VAR_INPUT
		(* Distance from the origin. *)
		radius : LREAL;
		(* Polar angle of this position in degrees [Â°]. *)
		phi : LREAL;
	END_VAR
END_METHOD


	(* Set the xy-coordinates of this position and the reference id. *)
	METHOD SetValuesXYReferenceId
	VAR_INPUT
		(* x-component of the position. *)
		x : LREAL;
		(* y-component of the position. *)
		y : LREAL;
		(* reference id of the position. *)
 {attribute 'GUID' := '18071995-0000-0000-0000-00000000000F'}
				ReferenceId : OTCID;
	END_VAR
END_METHOD


	(* Get the distance from the origin. *)
	METHOD GetRadius : LREAL
END_METHOD


	(* Get the polar angle scaled in degrees [Â°]. *)
	METHOD GetPhi : LREAL
END_METHOD


	(* Invert this position. *)
	METHOD Invert
END_METHOD


	(* Concatenate with a 2nd position. *)
	METHOD ConcatenateWith
	VAR_IN_OUT
		(* The 2nd position to concatenate with. *)
 {attribute 'GUID' := 'D1D75488-37B1-0155-53AF-A9A9BDBB4FFD'}
				position : PositionXY;
	END_VAR
END_METHOD


	(* Displace the components of this position. *)
	METHOD ShiftBy
	VAR_IN_OUT
		(* The displacement to shift by. *)
 {attribute 'GUID' := '619D5D7D-53EC-0B73-54D5-FB9C43AFDE82'}
				shift : TangentXY;
	END_VAR
END_METHOD


	(* Displace the components of this position. *)
	METHOD ShiftByXY
	VAR_INPUT
		(* Shift of the x-component of this position. *)
		dx : LREAL;
		(* Shift of the y-component of this position. *)
		dy : LREAL;
	END_VAR
END_METHOD


	PROPERTY x : LREAL
GET
END_GET
SET
END_SET
END_PROPERTY


	PROPERTY y : LREAL
GET
END_GET
SET
END_SET
END_PROPERTY


{attribute 'monitoring' := 'call'}
	PROPERTY ReferenceId : OTCID
GET
END_GET
SET
END_SET
END_PROPERTY

END_FUNCTION_BLOCK

// POUs/_Internal/Geometry3D

	{attribute 'c++_compatible'}
	{attribute 'external_name' := 'Geometry3D_GUID_56994EB0_AB4F_0BCB_4E0E_A36B53A3D853'}
	{attribute 'TcIecLibraryType'}
	{attribute 'no_explicit_call' :='do not call this POU directly'}
	{attribute 'no_assign'}
	(* Base class for all 3D Geo objects (simple geometries, container) *)
	FUNCTION_BLOCK Geometry3D EXTENDS IPlcGeometry3D


	(* Internal method *)
	METHOD FB_init : BOOL
	VAR_INPUT
		(*  if TRUE, the retain variables are initialized (warm start / cold start) *)
		bInitRetains : BOOL;
		(*  if TRUE, the instance afterwards gets moved into the copy code (online change) *)
		bInCopyCode : BOOL;
	END_VAR
END_METHOD


	(* Internal method *)
	{attribute 'hide'}
	METHOD FB_exit : BOOL
	VAR_INPUT
		(*  if TRUE, the exit method is called for exiting an instance that is copied afterwards (online change). *)
		bInCopyCode : BOOL;
	END_VAR
END_METHOD


	(* Set the local position of this geometry. *)
	METHOD SetDisplacement
	VAR_IN_OUT
		(* The position to set. *)
 {attribute 'GUID' := '4DF191CB-C971-05F9-659B-EBBADE382F22'}
				displacement : PositionSE3;
	END_VAR
END_METHOD


	(* Set the local position of this geometry. *)
	METHOD SetDisplacementXYZ
	VAR_INPUT
		(* x-component of the position. *)
		x : LREAL;
		(* y-component of the position. *)
		y : LREAL;
		(* z-component of the position. *)
		z : LREAL;
	END_VAR
END_METHOD


	(* Set the local position of this geometry. *)
	METHOD SetDisplacementX
	VAR_INPUT
		(* x-component of the position. *)
		x : LREAL;
	END_VAR
END_METHOD


	(* Set the local position of this geometry. *)
	METHOD SetDisplacementY
	VAR_INPUT
		(* y-component of the position. *)
		y : LREAL;
	END_VAR
END_METHOD


	(* Set the local position of this geometry. *)
	METHOD SetDisplacementZ
	VAR_INPUT
		(* z-component of the position. *)
		z : LREAL;
	END_VAR
END_METHOD


	(* Set the global position of this geometry. *)
	METHOD SetPosition
	VAR_IN_OUT
		(* The position to set. *)
 {attribute 'GUID' := '4DF191CB-C971-05F9-659B-EBBADE382F22'}
				position : PositionSE3;
	END_VAR
END_METHOD


	(* Set the global position of this geometry. *)
	METHOD SetPositionXYZ
	VAR_INPUT
		(* x-component of the position. *)
		x : LREAL;
		(* y-component of the position. *)
		y : LREAL;
		(* z-component of the position. *)
		z : LREAL;
	END_VAR
END_METHOD


	(* Set the global position of this geometry. *)
	METHOD SetPositionX
	VAR_INPUT
		(* x-component of the position. *)
		x : LREAL;
	END_VAR
END_METHOD


	(* Set the global position of this geometry. *)
	METHOD SetPositionY
	VAR_INPUT
		(* y-component of the position. *)
		y : LREAL;
	END_VAR
END_METHOD


	(* Set the global position of this geometry. *)
	METHOD SetPositionZ
	VAR_INPUT
		(* z-component of the position. *)
		z : LREAL;
	END_VAR
END_METHOD


	(* Set the coordinates of the orientation. *)
	METHOD SetRotationABC
	VAR_INPUT
		(* 1st rotation angle in degrees [Â°]. *)
		phi0 : LREAL;
		(* 2nd rotation angle in degrees [Â°]. *)
		phi1 : LREAL;
		(* 3rd rotation angle in degrees [Â°]. *)
		phi2 : LREAL;
	END_VAR
END_METHOD


	(* Set the coordinates of the orientation. *)
	METHOD SetRotationACB
	VAR_INPUT
		(* 1st rotation angle in degrees [Â°]. *)
		phi0 : LREAL;
		(* 2nd rotation angle in degrees [Â°]. *)
		phi1 : LREAL;
		(* 3rd rotation angle in degrees [Â°]. *)
		phi2 : LREAL;
	END_VAR
END_METHOD


	(* Set the coordinates of the orientation. *)
	METHOD SetRotationBCA
	VAR_INPUT
		(* 1st rotation angle in degrees [Â°]. *)
		phi0 : LREAL;
		(* 2nd rotation angle in degrees [Â°]. *)
		phi1 : LREAL;
		(* 3rd rotation angle in degrees [Â°]. *)
		phi2 : LREAL;
	END_VAR
END_METHOD


	(* Set the coordinates of the orientation. *)
	METHOD SetRotationBAC
	VAR_INPUT
		(* 1st rotation angle in degrees [Â°]. *)
		phi0 : LREAL;
		(* 2nd rotation angle in degrees [Â°]. *)
		phi1 : LREAL;
		(* 3rd rotation angle in degrees [Â°]. *)
		phi2 : LREAL;
	END_VAR
END_METHOD


	(* Set the coordinates of the orientation. *)
	METHOD SetRotationCAB
	VAR_INPUT
		(* 1st rotation angle in degrees [Â°]. *)
		phi0 : LREAL;
		(* 2nd rotation angle in degrees [Â°]. *)
		phi1 : LREAL;
		(* 3rd rotation angle in degrees [Â°]. *)
		phi2 : LREAL;
	END_VAR
END_METHOD


	(* Set the coordinates of the orientation. *)
	METHOD SetRotationCBA
	VAR_INPUT
		(* 1st rotation angle in degrees [Â°]. *)
		phi0 : LREAL;
		(* 2nd rotation angle in degrees [Â°]. *)
		phi1 : LREAL;
		(* 3rd rotation angle in degrees [Â°]. *)
		phi2 : LREAL;
	END_VAR
END_METHOD


	(* Set the coordinates of the orientation. *)
	METHOD SetRotationABA
	VAR_INPUT
		(* 1st rotation angle in degrees [Â°]. *)
		phi0 : LREAL;
		(* 2nd rotation angle in degrees [Â°]. *)
		phi1 : LREAL;
		(* 3rd rotation angle in degrees [Â°]. *)
		phi2 : LREAL;
	END_VAR
END_METHOD


	(* Set the coordinates of the orientation. *)
	METHOD SetRotationACA
	VAR_INPUT
		(* 1st rotation angle in degrees [Â°]. *)
		phi0 : LREAL;
		(* 2nd rotation angle in degrees [Â°]. *)
		phi1 : LREAL;
		(* 3rd rotation angle in degrees [Â°]. *)
		phi2 : LREAL;
	END_VAR
END_METHOD


	(* Set the coordinates of the orientation. *)
	METHOD SetRotationBCB
	VAR_INPUT
		(* 1st rotation angle in degrees [Â°]. *)
		phi0 : LREAL;
		(* 2nd rotation angle in degrees [Â°]. *)
		phi1 : LREAL;
		(* 3rd rotation angle in degrees [Â°]. *)
		phi2 : LREAL;
	END_VAR
END_METHOD


	(* Set the coordinates of the orientation. *)
	METHOD SetRotationBAB
	VAR_INPUT
		(* 1st rotation angle in degrees [Â°]. *)
		phi0 : LREAL;
		(* 2nd rotation angle in degrees [Â°]. *)
		phi1 : LREAL;
		(* 3rd rotation angle in degrees [Â°]. *)
		phi2 : LREAL;
	END_VAR
END_METHOD


	(* Set the coordinates of the orientation. *)
	METHOD SetRotationCAC
	VAR_INPUT
		(* 1st rotation angle in degrees [Â°]. *)
		phi0 : LREAL;
		(* 2nd rotation angle in degrees [Â°]. *)
		phi1 : LREAL;
		(* 3rd rotation angle in degrees [Â°]. *)
		phi2 : LREAL;
	END_VAR
END_METHOD


	(* Set the coordinates of the orientation. *)
	METHOD SetRotationCBC
	VAR_INPUT
		(* 1st rotation angle in degrees [Â°]. *)
		phi0 : LREAL;
		(* 2nd rotation angle in degrees [Â°]. *)
		phi1 : LREAL;
		(* 3rd rotation angle in degrees [Â°]. *)
		phi2 : LREAL;
	END_VAR
END_METHOD


	(* Get the global position of this geometry. *)
	METHOD GetDisplacement
	VAR_IN_OUT
		(* The current position of the geometry. *)
 {attribute 'GUID' := '4DF191CB-C971-05F9-659B-EBBADE382F22'}
				position : PositionSE3;
	END_VAR
END_METHOD


	(* Get the global x-component of this geometry. *)
	METHOD GetDisplacementX : LREAL
END_METHOD


	(* Get the global y-component of this geometry. *)
	METHOD GetDisplacementY : LREAL
END_METHOD


	(* Get the global z-component of this geometry. *)
	METHOD GetDisplacementZ : LREAL
END_METHOD


	(* Get the local direction of the local x-axis. *)
	METHOD GetLocalX
	VAR_IN_OUT
		(* The local x-direction of this orientation. *)
 {attribute 'GUID' := 'B2E383A0-A70D-05BB-6EF1-4EF1FE579E25'}
				localX : Tangent3D;
	END_VAR
END_METHOD


	(* Get the local direction of the local y-axis. *)
	METHOD GetLocalY
	VAR_IN_OUT
		(* The local y-direction of this orientation. *)
 {attribute 'GUID' := 'B2E383A0-A70D-05BB-6EF1-4EF1FE579E25'}
				localY : Tangent3D;
	END_VAR
END_METHOD


	(* Get the local direction of the local z-axis. *)
	METHOD GetLocalZ
	VAR_IN_OUT
		(* The local z-direction of this orientation. *)
 {attribute 'GUID' := 'B2E383A0-A70D-05BB-6EF1-4EF1FE579E25'}
				localZ : Tangent3D;
	END_VAR
END_METHOD


	(* Get the global position of this geometry. *)
	METHOD GetPosition
	VAR_IN_OUT
		(* The current position of the geometry. *)
 {attribute 'GUID' := '4DF191CB-C971-05F9-659B-EBBADE382F22'}
				position : PositionSE3;
	END_VAR
END_METHOD


	(* Get the global x-component of this geometry. *)
	METHOD GetPositionX : LREAL
END_METHOD


	(* Get the global y-component of this geometry. *)
	METHOD GetPositionY : LREAL
END_METHOD


	(* Get the global z-component of this geometry. *)
	METHOD GetPositionZ : LREAL
END_METHOD


	(* Get the global direction of the local x-axis. *)
	METHOD GetDirectionX
	VAR_IN_OUT
		(* The local x-direction of this orientation. *)
 {attribute 'GUID' := 'B2E383A0-A70D-05BB-6EF1-4EF1FE579E25'}
				localX : Tangent3D;
	END_VAR
END_METHOD


	(* Get the global direction of the local y-axis. *)
	METHOD GetDirectionY
	VAR_IN_OUT
		(* The local y-direction of this orientation. *)
 {attribute 'GUID' := 'B2E383A0-A70D-05BB-6EF1-4EF1FE579E25'}
				localY : Tangent3D;
	END_VAR
END_METHOD


	(* Get the global direction of the local z-axis. *)
	METHOD GetDirectionZ
	VAR_IN_OUT
		(* The local z-direction of this orientation. *)
 {attribute 'GUID' := 'B2E383A0-A70D-05BB-6EF1-4EF1FE579E25'}
				localZ : Tangent3D;
	END_VAR
END_METHOD


	(* Displace the components of this position. The shift is applied within the local coordinate frame. *)
	METHOD StepByLocal
	VAR_IN_OUT
		(* The displacement to shift by. *)
 {attribute 'GUID' := '41AC0F4B-9126-0537-6401-E7160585CD6C'}
				shift : Tangent6D;
	END_VAR
END_METHOD


	(* Apply a local step in respect to the local coordinate frame without changing the orientation. *)
	METHOD StepByLocalXYZ
	VAR_INPUT
		(* The displacement within the local x-direction. *)
		dx : LREAL;
		(* The displacement within the local y-direction. *)
		dy : LREAL;
		(* The displacement within the local z-direction. *)
		dz : LREAL;
	END_VAR
END_METHOD


	(* Displace the components of this position. *)
	METHOD ShiftBy
	VAR_IN_OUT
		(* Shift vector to displace by. *)
 {attribute 'GUID' := 'B2E383A0-A70D-05BB-6EF1-4EF1FE579E25'}
				shift : Tangent3D;
	END_VAR
END_METHOD


	(* Displace the components of this position. *)
	METHOD ShiftByXYZ
	VAR_INPUT
		(* Shift of the x-component of this position. *)
		dx : LREAL;
		(* Shift of the y-component of this position. *)
		dy : LREAL;
		(* Shift of the z-component of this position. *)
		dz : LREAL;
	END_VAR
END_METHOD


	(* Rotate around an arbitrary local axis. The turn angle is given by the length of the axis. *)
	METHOD TurnBy
	VAR_IN_OUT
		(* The axis of rotation. Its length represents the angle of rotation in degrees [Â°]. *)
 {attribute 'GUID' := '40BB739E-8B51-070D-548D-A1BF22EE7364'}
				axis : TangentABC;
	END_VAR
END_METHOD


	(* Rotation around the local x-axis. *)
	METHOD TurnByA
	VAR_INPUT
		(* The angle to rotate by in degrees [Â°]. *)
		da : LREAL;
	END_VAR
END_METHOD


	(* Rotation around the local y-axis. *)
	METHOD TurnByB
	VAR_INPUT
		(* The angle to rotate by in degrees [Â°]. *)
		db : LREAL;
	END_VAR
END_METHOD


	(* Rotation around the local z-axis. *)
	METHOD TurnByC
	VAR_INPUT
		(* The angle to rotate by in degrees [Â°]. *)
		dc : LREAL;
	END_VAR
END_METHOD


	PROPERTY phi0 : LREAL
GET
END_GET
SET
END_SET
END_PROPERTY


	PROPERTY phi1 : LREAL
GET
END_GET
SET
END_SET
END_PROPERTY


	PROPERTY phi2 : LREAL
GET
END_GET
SET
END_SET
END_PROPERTY


	PROPERTY Convention : E_RotationCoordinates
GET
END_GET
SET
END_SET
END_PROPERTY

END_FUNCTION_BLOCK

// POUs/Spatial/Positions/PositionSE3

	{attribute 'c++_compatible'}
	{attribute 'external_name' := 'PositionSE3_GUID_4DF191CB_C971_05F9_659B_EBBADE382F22'}
	{attribute 'TcIecLibraryType'}
	{attribute 'no_explicit_call' :='do not call this POU directly'}
	{attribute 'no_assign'}
	(* 6D position containing position and orientation. All angles in degrees [Ã‚Â°]. *)
	FUNCTION_BLOCK PositionSE3 EXTENDS IPlcGeometry3D


	(* Internal method *)
	{attribute 'hide'}
	METHOD FB_init : BOOL
	VAR_INPUT
		(*  if TRUE, the retain variables are initialized (warm start / cold start) *)
		bInitRetains : BOOL;
		(*  if TRUE, the instance afterwards gets moved into the copy code (online change) *)
		bInCopyCode : BOOL;
	END_VAR
END_METHOD


	(* Internal method *)
	{attribute 'hide'}
	METHOD FB_exit : BOOL
	VAR_INPUT
		(*  if TRUE, the exit method is called for exiting an instance that is copied afterwards (online change). *)
		bInCopyCode : BOOL;
	END_VAR
END_METHOD


	(* Set the components of this position to '0.0'. *)
	METHOD SetZero
END_METHOD


	(* Set the components of this position. *)
	METHOD SetValues
	VAR_IN_OUT
		(* The position values to set. *)
 {attribute 'GUID' := '4DF191CB-C971-05F9-659B-EBBADE382F22'}
				positionSE3 : PositionSE3;
	END_VAR
END_METHOD


	(* Set the components of this position. *)
	METHOD SetValuesXYZ
	VAR_INPUT
		(* x-component of the position. *)
		x : LREAL;
		(* y-component of the position. *)
		y : LREAL;
		(* z-component of the position. *)
		z : LREAL;
	END_VAR
END_METHOD


	(* Set the components of this position in cylindric coordinates. *)
	METHOD SetValuesRPZ
	VAR_INPUT
		(* Distance from the z-axis. *)
		radius : LREAL;
		(* Polar angle in degrees [Ã‚Â°]. *)
		phi : LREAL;
		(* z-component of the position. *)
		z : LREAL;
	END_VAR
END_METHOD


	(* Set the components of this position in spherical coordinates. *)
	METHOD SetValuesRTP
	VAR_INPUT
		(* Distance from the origin. *)
		_r : LREAL;
		(* Azimuthal angle in degrees [Ã‚Â°]. *)
		t : LREAL;
		(* Polar angle in degrees [Ã‚Â°]. *)
		p : LREAL;
	END_VAR
END_METHOD


	(* Set the coordinates of the orientation. *)
	METHOD SetValuesABC
	VAR_INPUT
		(* 1st rotation angle in degrees [Ã‚Â°]. *)
		phi0 : LREAL;
		(* 2nd rotation angle in degrees [Ã‚Â°]. *)
		phi1 : LREAL;
		(* 3rd rotation angle in degrees [Ã‚Â°]. *)
		phi2 : LREAL;
	END_VAR
END_METHOD


	(* Set the coordinates of the orientation. *)
	METHOD SetValuesACB
	VAR_INPUT
		(* 1st rotation angle in degrees [Ã‚Â°]. *)
		phi0 : LREAL;
		(* 2nd rotation angle in degrees [Ã‚Â°]. *)
		phi1 : LREAL;
		(* 3rd rotation angle in degrees [Ã‚Â°]. *)
		phi2 : LREAL;
	END_VAR
END_METHOD


	(* Set the coordinates of the orientation. *)
	METHOD SetValuesBCA
	VAR_INPUT
		(* 1st rotation angle in degrees [Ã‚Â°]. *)
		phi0 : LREAL;
		(* 2nd rotation angle in degrees [Ã‚Â°]. *)
		phi1 : LREAL;
		(* 3rd rotation angle in degrees [Ã‚Â°]. *)
		phi2 : LREAL;
	END_VAR
END_METHOD


	(* Set the coordinates of the orientation. *)
	METHOD SetValuesBAC
	VAR_INPUT
		(* 1st rotation angle in degrees [Ã‚Â°]. *)
		phi0 : LREAL;
		(* 2nd rotation angle in degrees [Ã‚Â°]. *)
		phi1 : LREAL;
		(* 3rd rotation angle in degrees [Ã‚Â°]. *)
		phi2 : LREAL;
	END_VAR
END_METHOD


	(* Set the coordinates of the orientation. *)
	METHOD SetValuesCAB
	VAR_INPUT
		(* 1st rotation angle in degrees [Ã‚Â°]. *)
		phi0 : LREAL;
		(* 2nd rotation angle in degrees [Ã‚Â°]. *)
		phi1 : LREAL;
		(* 3rd rotation angle in degrees [Ã‚Â°]. *)
		phi2 : LREAL;
	END_VAR
END_METHOD


	(* Set the coordinates of the orientation. *)
	METHOD SetValuesCBA
	VAR_INPUT
		(* 1st rotation angle in degrees [Ã‚Â°]. *)
		phi0 : LREAL;
		(* 2nd rotation angle in degrees [Ã‚Â°]. *)
		phi1 : LREAL;
		(* 3rd rotation angle in degrees [Ã‚Â°]. *)
		phi2 : LREAL;
	END_VAR
END_METHOD


	(* Set the coordinates of the orientation. *)
	METHOD SetValuesABA
	VAR_INPUT
		(* 1st rotation angle in degrees [Ã‚Â°]. *)
		phi0 : LREAL;
		(* 2nd rotation angle in degrees [Ã‚Â°]. *)
		phi1 : LREAL;
		(* 3rd rotation angle in degrees [Ã‚Â°]. *)
		phi2 : LREAL;
	END_VAR
END_METHOD


	(* Set the coordinates of the orientation. *)
	METHOD SetValuesACA
	VAR_INPUT
		(* 1st rotation angle in degrees [Ã‚Â°]. *)
		phi0 : LREAL;
		(* 2nd rotation angle in degrees [Ã‚Â°]. *)
		phi1 : LREAL;
		(* 3rd rotation angle in degrees [Ã‚Â°]. *)
		phi2 : LREAL;
	END_VAR
END_METHOD


	(* Set the coordinates of the orientation. *)
	METHOD SetValuesBCB
	VAR_INPUT
		(* 1st rotation angle in degrees [Ã‚Â°]. *)
		phi0 : LREAL;
		(* 2nd rotation angle in degrees [Ã‚Â°]. *)
		phi1 : LREAL;
		(* 3rd rotation angle in degrees [Ã‚Â°]. *)
		phi2 : LREAL;
	END_VAR
END_METHOD


	(* Set the coordinates of the orientation. *)
	METHOD SetValuesBAB
	VAR_INPUT
		(* 1st rotation angle in degrees [Ã‚Â°]. *)
		phi0 : LREAL;
		(* 2nd rotation angle in degrees [Ã‚Â°]. *)
		phi1 : LREAL;
		(* 3rd rotation angle in degrees [Ã‚Â°]. *)
		phi2 : LREAL;
	END_VAR
END_METHOD


	(* Set the coordinates of the orientation. *)
	METHOD SetValuesCAC
	VAR_INPUT
		(* 1st rotation angle in degrees [Ã‚Â°]. *)
		phi0 : LREAL;
		(* 2nd rotation angle in degrees [Ã‚Â°]. *)
		phi1 : LREAL;
		(* 3rd rotation angle in degrees [Ã‚Â°]. *)
		phi2 : LREAL;
	END_VAR
END_METHOD


	(* Set the coordinates of the orientation. *)
	METHOD SetValuesCBC
	VAR_INPUT
		(* 1st rotation angle in degrees [Ã‚Â°]. *)
		phi0 : LREAL;
		(* 2nd rotation angle in degrees [Ã‚Â°]. *)
		phi1 : LREAL;
		(* 3rd rotation angle in degrees [Ã‚Â°]. *)
		phi2 : LREAL;
	END_VAR
END_METHOD


	(* Get the direction of the local x-axis. *)
	METHOD GetDirectionX
	VAR_IN_OUT
		(* The local x-direction of this orientation. *)
 {attribute 'GUID' := 'B2E383A0-A70D-05BB-6EF1-4EF1FE579E25'}
				localX : Tangent3D;
	END_VAR
END_METHOD


	(* Get the direction of the local y-axis. *)
	METHOD GetDirectionY
	VAR_IN_OUT
		(* The local y-direction of this orientation. *)
 {attribute 'GUID' := 'B2E383A0-A70D-05BB-6EF1-4EF1FE579E25'}
				localY : Tangent3D;
	END_VAR
END_METHOD


	(* Get the direction of the local z-axis. *)
	METHOD GetDirectionZ
	VAR_IN_OUT
		(* The local z-direction of this orientation. *)
 {attribute 'GUID' := 'B2E383A0-A70D-05BB-6EF1-4EF1FE579E25'}
				localZ : Tangent3D;
	END_VAR
END_METHOD


	(* Invert this position. *)
	METHOD Invert
END_METHOD


	(* Applies a transformation (shift, rotation) to this position *)
	METHOD ConcatenateWith
	VAR_IN_OUT
		(* transformation (shift, rotation) to be applied *)
 {attribute 'GUID' := '4DF191CB-C971-05F9-659B-EBBADE382F22'}
				position : PositionSE3;
	END_VAR
END_METHOD


	(* Displace the components of this position. The shift is applied within the local coordinate frame. *)
	METHOD StepByLocal
	VAR_IN_OUT
		(* The displacement to shift by. *)
 {attribute 'GUID' := '41AC0F4B-9126-0537-6401-E7160585CD6C'}
				shift : Tangent6D;
	END_VAR
END_METHOD


	(* Apply a local step in respect to the local coordinate frame without changing the orientation. *)
	METHOD StepByLocalXYZ
	VAR_INPUT
		(* The displacement within the local x-direction. *)
		dx : LREAL;
		(* The displacement within the local y-direction. *)
		dy : LREAL;
		(* The displacement within the local z-direction. *)
		dz : LREAL;
	END_VAR
END_METHOD


	(* Displace the components of this position. *)
	METHOD ShiftBy
	VAR_IN_OUT
		(* Shift vector to displace by. *)
 {attribute 'GUID' := 'B2E383A0-A70D-05BB-6EF1-4EF1FE579E25'}
				shift : Tangent3D;
	END_VAR
END_METHOD


	(* Displace the components of this position. *)
	METHOD ShiftByXYZ
	VAR_INPUT
		(* Shift of the x-component of this position. *)
		dx : LREAL;
		(* Shift of the y-component of this position. *)
		dy : LREAL;
		(* Shift of the z-component of this position. *)
		dz : LREAL;
	END_VAR
END_METHOD


	(* Rotate around an arbitrary local axis. The turn angle is given by the length of the axis. *)
	METHOD TurnBy
	VAR_IN_OUT
		(* The axis of rotation. Its length represents the angle of rotation in degrees [Ã‚Â°]. *)
 {attribute 'GUID' := '40BB739E-8B51-070D-548D-A1BF22EE7364'}
				axis : TangentABC;
	END_VAR
END_METHOD


	(* Rotation around the local x-axis. *)
	METHOD TurnByA
	VAR_INPUT
		(* The angle to rotate by in degrees [Ã‚Â°]. *)
		da : LREAL;
	END_VAR
END_METHOD


	(* Rotation around the local y-axis. *)
	METHOD TurnByB
	VAR_INPUT
		(* The angle to rotate by in degrees [Ã‚Â°]. *)
		db : LREAL;
	END_VAR
END_METHOD


	(* Rotation around the local z-axis. *)
	METHOD TurnByC
	VAR_INPUT
		(* The angle to rotate by in degrees [Ã‚Â°]. *)
		dc : LREAL;
	END_VAR
END_METHOD


	(* Rotate a Position3D according to this transformation. *)
	METHOD Transform
	VAR_IN_OUT
		(* Position to transform. *)
 {attribute 'GUID' := '6D9DE39A-582F-0FB5-796C-F5BBE97EF7B7'}
				position : Position3D;
	END_VAR
END_METHOD


	PROPERTY x : LREAL
GET
END_GET
SET
END_SET
END_PROPERTY


	PROPERTY y : LREAL
GET
END_GET
SET
END_SET
END_PROPERTY


	PROPERTY z : LREAL
GET
END_GET
SET
END_SET
END_PROPERTY


	PROPERTY phi0 : LREAL
GET
END_GET
SET
END_SET
END_PROPERTY


	PROPERTY phi1 : LREAL
GET
END_GET
SET
END_SET
END_PROPERTY


	PROPERTY phi2 : LREAL
GET
END_GET
SET
END_SET
END_PROPERTY


	PROPERTY Convention : E_RotationCoordinates
GET
END_GET
SET
END_SET
END_PROPERTY

END_FUNCTION_BLOCK

// POUs/Spatial/Tangents/Tangent3D

	{attribute 'c++_compatible'}
	{attribute 'external_name' := 'Tangent3D_GUID_B2E383A0_A70D_05BB_6EF1_4EF1FE579E25'}
	{attribute 'TcIecLibraryType'}
	{attribute 'no_explicit_call' :='do not call this POU directly'}
	{attribute 'no_assign'}
	(* A Cartesian direction to describe a displacement or velocity in the 3D-Cartesian space. *)
	FUNCTION_BLOCK Tangent3D
	VAR
		(* x-component of the tangent *)
		dx : LREAL;
		(* y-component of the tangent *)
		dy : LREAL;
		(* z-component of the tangent *)
		dz : LREAL;
		 {attribute 'hide'}
		_reserved1 : ARRAY [1..88] OF USINT;
	END_VAR


	(* Internal method *)
	{attribute 'hide'}
	METHOD FB_init : BOOL
	VAR_INPUT
		(*  if TRUE, the retain variables are initialized (warm start / cold start) *)
		bInitRetains : BOOL;
		(*  if TRUE, the instance afterwards gets moved into the copy code (online change) *)
		bInCopyCode : BOOL;
	END_VAR
END_METHOD


	(* Internal method *)
	{attribute 'hide'}
	METHOD FB_exit : BOOL
	VAR_INPUT
		(*  if TRUE, the exit method is called for exiting an instance that is copied afterwards (online change). *)
		bInCopyCode : BOOL;
	END_VAR
END_METHOD


	(* Set the components of this tangent to '0.0'. *)
	METHOD SetZero
END_METHOD


	(* Set the components of this tangent. *)
	METHOD SetValues
	VAR_IN_OUT
		(* The tangent values to set. *)
 {attribute 'GUID' := 'B2E383A0-A70D-05BB-6EF1-4EF1FE579E25'}
				tangent3D : Tangent3D;
	END_VAR
END_METHOD


	(* Set the components of this tangent. *)
	METHOD SetValuesXYZ
	VAR_INPUT
		(* x-component of the tangent. *)
		x : LREAL;
		(* y-component of the tangent. *)
		y : LREAL;
		(* z-component of the tangent. *)
		z : LREAL;
	END_VAR
END_METHOD


	(* Check if all components of this tangent are within a tolerance from zero. *)
	METHOD IsZero : BOOL
	VAR_INPUT
		(* The tolerance threshold for each of the components. *)
		tolerance : LREAL;
	END_VAR
END_METHOD


	(* Get the Euclidean length of this tangent vector. *)
	METHOD GetLength : LREAL
END_METHOD


	(* Get the normalized direction to this tangent vector. *)
	METHOD GetDirection
	VAR_IN_OUT
		(* The normalized direction vector. *)
 {attribute 'GUID' := 'B2E383A0-A70D-05BB-6EF1-4EF1FE579E25'}
				direction : Tangent3D;
	END_VAR
END_METHOD


	(* Add a 2nd tangent vector to this one. *)
	METHOD AddBy
	VAR_IN_OUT
		(* The tangent vector to add. *)
 {attribute 'GUID' := 'B2E383A0-A70D-05BB-6EF1-4EF1FE579E25'}
				shift : Tangent3D;
	END_VAR
END_METHOD


	(* Add values to each of the components of this tangent vector. *)
	METHOD AddByXYZ
	VAR_INPUT
		(* Value to add to the x-component. *)
		dx : LREAL;
		(* Value to add to the y-component. *)
		dy : LREAL;
		(* Value to add to the z-component. *)
		dz : LREAL;
	END_VAR
END_METHOD


	(* Subtract a 2nd tangent vector from this one. *)
	METHOD SubtractBy
	VAR_IN_OUT
		(* The tangent vector to subtract. *)
 {attribute 'GUID' := 'B2E383A0-A70D-05BB-6EF1-4EF1FE579E25'}
				shift : Tangent3D;
	END_VAR
END_METHOD


	(* Subtract values from each of the components of this tangent vector. *)
	METHOD SubtractByXYZ
	VAR_INPUT
		(* Value to subtract from the x-component. *)
		dx : LREAL;
		(* Value to subtract from the y-component. *)
		dy : LREAL;
		(* Value to subtract from the z-component. *)
		dz : LREAL;
	END_VAR
END_METHOD


	(* Multiply the components of this tangent vector by a number. *)
	METHOD MultiplyBy
	VAR_INPUT
		(* The number to scale this tangent by. *)
		scale : LREAL;
	END_VAR
END_METHOD


	(* Divide the components of this tangent vector by a number. *)
	METHOD DivideBy
	VAR_INPUT
		(* The number to divide this tangent by. *)
		scale : LREAL;
	END_VAR
END_METHOD


	(* Normalize this tangent. *)
	METHOD Normalize
END_METHOD


	PROPERTY x : LREAL
GET
END_GET
SET
END_SET
END_PROPERTY


	PROPERTY y : LREAL
GET
END_GET
SET
END_SET
END_PROPERTY


	PROPERTY z : LREAL
GET
END_GET
SET
END_SET
END_PROPERTY

END_FUNCTION_BLOCK

// POUs/Spatial/Tangents/Tangent6D

	{attribute 'c++_compatible'}
	{attribute 'external_name' := 'Tangent6D_GUID_41AC0F4B_9126_0537_6401_E7160585CD6C'}
	{attribute 'TcIecLibraryType'}
	{attribute 'no_explicit_call' :='do not call this POU directly'}
	{attribute 'no_assign'}
	(* An Euclidean direction to describe
				  a displacement or velocity in the local 3D-Cartesian space
				  with additional angular displacement information. *)
	FUNCTION_BLOCK Tangent6D
	VAR
	END_VAR


	(* Internal method *)
	{attribute 'hide'}
	METHOD FB_init : BOOL
	VAR_INPUT
		(*  if TRUE, the retain variables are initialized (warm start / cold start) *)
		bInitRetains : BOOL;
		(*  if TRUE, the instance afterwards gets moved into the copy code (online change) *)
		bInCopyCode : BOOL;
	END_VAR
END_METHOD


	(* Internal method *)
	{attribute 'hide'}
	METHOD FB_exit : BOOL
	VAR_INPUT
		(*  if TRUE, the exit method is called for exiting an instance that is copied afterwards (online change). *)
		bInCopyCode : BOOL;
	END_VAR
END_METHOD

END_FUNCTION_BLOCK

// POUs/Spatial/Tangents/TangentABC

	{attribute 'c++_compatible'}
	{attribute 'external_name' := 'TangentABC_GUID_40BB739E_8B51_070D_548D_A1BF22EE7364'}
	{attribute 'TcIecLibraryType'}
	{attribute 'no_explicit_call' :='do not call this POU directly'}
	{attribute 'no_assign'}
	(* A 3-dimensional angular velocity or rotation axis, all components are scaled in degrees [Â°]. *)
	FUNCTION_BLOCK TangentABC
	VAR
		(* a-component of the tangent *)
		da : LREAL;
		(* b-component of the tangent *)
		db : LREAL;
		(* c-component of the tangent *)
		dc : LREAL;
		 {attribute 'hide'}
		_reserved1 : ARRAY [1..88] OF USINT;
	END_VAR


	(* Internal method *)
	{attribute 'hide'}
	METHOD FB_init : BOOL
	VAR_INPUT
		(*  if TRUE, the retain variables are initialized (warm start / cold start) *)
		bInitRetains : BOOL;
		(*  if TRUE, the instance afterwards gets moved into the copy code (online change) *)
		bInCopyCode : BOOL;
	END_VAR
END_METHOD


	(* Internal method *)
	{attribute 'hide'}
	METHOD FB_exit : BOOL
	VAR_INPUT
		(*  if TRUE, the exit method is called for exiting an instance that is copied afterwards (online change). *)
		bInCopyCode : BOOL;
	END_VAR
END_METHOD


	(* Set the components of this tangent to '0.0'. *)
	METHOD SetZero
END_METHOD


	(* Set the components of this tangent. *)
	METHOD SetValues
	VAR_IN_OUT
		(* The tangent values to set. *)
 {attribute 'GUID' := '40BB739E-8B51-070D-548D-A1BF22EE7364'}
				tangentABC : TangentABC;
	END_VAR
END_METHOD


	(* Set the components of this tangent. *)
	METHOD SetValuesABC
	VAR_INPUT
		(* a-component of the tangent in degrees [Â°]. *)
		x : LREAL;
		(* b-component of the tangent in degrees [Â°]. *)
		y : LREAL;
		(* c-component of the tangent in degrees [Â°]. *)
		z : LREAL;
	END_VAR
END_METHOD


	(* Check if all components of this tangent are within a tolerance from zero. *)
	METHOD IsZero : BOOL
	VAR_INPUT
		(* The tolerance threshold for each of the components. *)
		tolerance : LREAL;
	END_VAR
END_METHOD


	(* Get the Euclidean length of this tangent vector. *)
	METHOD GetLength : LREAL
END_METHOD


	(* Add a 2nd tangent vector to this one. *)
	METHOD AddBy
	VAR_IN_OUT
		(* The tangent vector to add. *)
 {attribute 'GUID' := '40BB739E-8B51-070D-548D-A1BF22EE7364'}
				shift : TangentABC;
	END_VAR
END_METHOD


	(* Add values to each of the components of this tangent vector. *)
	METHOD AddByABC
	VAR_INPUT
		(* Value to add to the a-component. *)
		da : LREAL;
		(* Value to add to the b-component. *)
		db : LREAL;
		(* Value to add to the c-component. *)
		dc : LREAL;
	END_VAR
END_METHOD


	(* Subtract a 2nd tangent vector from this one. *)
	METHOD SubtractBy
	VAR_IN_OUT
		(* The tangent vector to subtract. *)
 {attribute 'GUID' := '40BB739E-8B51-070D-548D-A1BF22EE7364'}
				shift : TangentABC;
	END_VAR
END_METHOD


	(* Subtract values from each of the components of this tangent vector. *)
	METHOD SubtractByABC
	VAR_INPUT
		(* Value to subtract from the a-component. *)
		da : LREAL;
		(* Value to subtract from the b-component. *)
		db : LREAL;
		(* Value to subtract from the c-component. *)
		dc : LREAL;
	END_VAR
END_METHOD


	(* Multiply the components of this tangent vector by a number. *)
	METHOD MultiplyBy
	VAR_INPUT
		(* The number to scale this tangent by. *)
		scale : LREAL;
	END_VAR
END_METHOD


	PROPERTY a : LREAL
GET
END_GET
SET
END_SET
END_PROPERTY


	PROPERTY b : LREAL
GET
END_GET
SET
END_SET
END_PROPERTY


	PROPERTY c : LREAL
GET
END_GET
SET
END_SET
END_PROPERTY

END_FUNCTION_BLOCK

// POUs/Spatial/Positions/Position3D

	{attribute 'c++_compatible'}
	{attribute 'external_name' := 'Position3D_GUID_6D9DE39A_582F_0FB5_796C_F5BBE97EF7B7'}
	{attribute 'TcIecLibraryType'}
	{attribute 'no_explicit_call' :='do not call this POU directly'}
	{attribute 'no_assign'}
	(* Position in the 3D Cartesian space. *)
	FUNCTION_BLOCK Position3D EXTENDS IPlcGeometry3D


	(* Internal method *)
	{attribute 'hide'}
	METHOD FB_init : BOOL
	VAR_INPUT
		(*  if TRUE, the retain variables are initialized (warm start / cold start) *)
		bInitRetains : BOOL;
		(*  if TRUE, the instance afterwards gets moved into the copy code (online change) *)
		bInCopyCode : BOOL;
	END_VAR
END_METHOD


	(* Internal method *)
	{attribute 'hide'}
	METHOD FB_exit : BOOL
	VAR_INPUT
		(*  if TRUE, the exit method is called for exiting an instance that is copied afterwards (online change). *)
		bInCopyCode : BOOL;
	END_VAR
END_METHOD


	(* Set the components of this vector to '0.0'. *)
	METHOD SetZero
END_METHOD


	(* Set the components of this position. *)
	METHOD SetValues
	VAR_IN_OUT
		(* The position values to set. *)
 {attribute 'GUID' := '6D9DE39A-582F-0FB5-796C-F5BBE97EF7B7'}
				position3D : Position3D;
	END_VAR
END_METHOD


	(* Set the components of this position. *)
	METHOD SetValuesXYZ
	VAR_INPUT
		(* x-component of the position. *)
		x : LREAL;
		(* y-component of the position. *)
		y : LREAL;
		(* z-component of the position. *)
		z : LREAL;
	END_VAR
END_METHOD


	(* Set the components of this position in cylindric coordinates. *)
	METHOD SetValuesRPZ
	VAR_INPUT
		(* Distance from the z-axis. *)
		radius : LREAL;
		(* Polar angle in degrees [Â°]. *)
		phi : LREAL;
		(* z-component of the position. *)
		z : LREAL;
	END_VAR
END_METHOD


	(* Set the components of this position in spherical coordinates. *)
	METHOD SetValuesRTP
	VAR_INPUT
		(* Distance from the origin. *)
		_r : LREAL;
		(* Azimuthal angle in degrees [Â°]. *)
		t : LREAL;
		(* Polar angle in degrees [Â°]. *)
		p : LREAL;
	END_VAR
END_METHOD


	(* Invert this position. *)
	METHOD Invert
END_METHOD


	(* Concatenate with a 2nd position. *)
	METHOD ConcatenateWith
	VAR_IN_OUT
		(* The 2nd position to concatenate with. *)
 {attribute 'GUID' := '6D9DE39A-582F-0FB5-796C-F5BBE97EF7B7'}
				position : Position3D;
	END_VAR
END_METHOD


	(* Displace the components of this position. *)
	METHOD ShiftBy
	VAR_IN_OUT
		(* The displacement to shift by. *)
 {attribute 'GUID' := 'B2E383A0-A70D-05BB-6EF1-4EF1FE579E25'}
				shift : Tangent3D;
	END_VAR
END_METHOD


	(* Displace the components of this position. *)
	METHOD ShiftByXYZ
	VAR_INPUT
		(* Shift of the x-component of this position. *)
		dx : LREAL;
		(* Shift of the y-component of this position. *)
		dy : LREAL;
		(* Shift of the z-component of this position. *)
		dz : LREAL;
	END_VAR
END_METHOD


	PROPERTY x : LREAL
GET
END_GET
SET
END_SET
END_PROPERTY


	PROPERTY y : LREAL
GET
END_GET
SET
END_SET
END_PROPERTY


	PROPERTY z : LREAL
GET
END_GET
SET
END_SET
END_PROPERTY

END_FUNCTION_BLOCK

// POUs/_Internal/IPlcPath2D

	{attribute 'c++_compatible'}
	{attribute 'external_name' := 'IPlcPath2D_GUID_30F67076_9DAC_07B9_5BCE_37111E6553BD'}
	{attribute 'TcIecLibraryType'}
	{attribute 'no_explicit_call' :='do not call this POU directly'}
	{attribute 'no_assign'}
	(* Internal representation of a path in the planar space. *)
	FUNCTION_BLOCK IPlcPath2D EXTENDS IPlcGeometry2D


	(* Internal method *)
	{attribute 'hide'}
	METHOD FB_init : BOOL
	VAR_INPUT
		(*  if TRUE, the retain variables are initialized (warm start / cold start) *)
		bInitRetains : BOOL;
		(*  if TRUE, the instance afterwards gets moved into the copy code (online change) *)
		bInCopyCode : BOOL;
	END_VAR
END_METHOD


	(* Internal method *)
	{attribute 'hide'}
	METHOD FB_exit : BOOL
	VAR_INPUT
		(*  if TRUE, the exit method is called for exiting an instance that is copied afterwards (online change). *)
		bInCopyCode : BOOL;
	END_VAR
END_METHOD


	(* Connect start and end position.
				      A smooth transition is added as long as start and end positin are not identical.
				      This operation finalizes this path definition and locks it against further modifications. *)
	METHOD CloseLoop
END_METHOD


	(* Empty all current path definitions and reset the path back to an empty state. *)
	METHOD Clear
END_METHOD


	(* Get the Euclidean length of the entire path chain. *)
	METHOD GetLength : LREAL
END_METHOD


	(* Check whether the start and end of the path chain are C2-continuously connected to each other. *)
	METHOD IsClosedLoop : BOOL
END_METHOD


	(* Check whether the path is self colliding. *)
	METHOD IsSelfColliding : BOOL
END_METHOD


	(* Calculate the arclength value where the path is closest to a geometry. *)
	METHOD GetArcLength_ClosestTo : LREAL
	VAR_IN_OUT
		(* The geometry to check the arc length for. *)
 {attribute 'GUID' := '0554E5C0-4687-0E31-67FE-D976C958432A'}
				geometry : IPlcGeometry2D;
	END_VAR
END_METHOD

END_FUNCTION_BLOCK

// POUs/_Internal/IPlcPath3D

	{attribute 'c++_compatible'}
	{attribute 'external_name' := 'IPlcPath3D_GUID_0696BF06_B4CF_0A9B_4B8B_86074F0A8B0C'}
	{attribute 'TcIecLibraryType'}
	{attribute 'no_explicit_call' :='do not call this POU directly'}
	{attribute 'no_assign'}
	(* Internal representation of a path in the planar space. *)
	FUNCTION_BLOCK IPlcPath3D EXTENDS IPlcGeometry3D


	(* Internal method *)
	{attribute 'hide'}
	METHOD FB_init : BOOL
	VAR_INPUT
		(*  if TRUE, the retain variables are initialized (warm start / cold start) *)
		bInitRetains : BOOL;
		(*  if TRUE, the instance afterwards gets moved into the copy code (online change) *)
		bInCopyCode : BOOL;
	END_VAR
END_METHOD


	(* Internal method *)
	{attribute 'hide'}
	METHOD FB_exit : BOOL
	VAR_INPUT
		(*  if TRUE, the exit method is called for exiting an instance that is copied afterwards (online change). *)
		bInCopyCode : BOOL;
	END_VAR
END_METHOD


	(* Connect start and end position.
				      A smooth transition is added as long as start and end positin are not identical.
				      This operation finalizes this path definition and locks it against further modifications. *)
	METHOD CloseLoop
END_METHOD


	(* Empty all current path definitions and reset the path back to an empty state. *)
	METHOD Clear
END_METHOD


	(* Get the Euclidean length of the entire path chain. *)
	METHOD GetLength : LREAL
END_METHOD


	(* Check whether the start and end of the path chain are C2-continuously connected to each other. *)
	METHOD IsClosedLoop : BOOL
END_METHOD


	(* Check whether the path is self colliding. *)
	METHOD IsSelfColliding : BOOL
END_METHOD


	(* Calculate the arclength value where the path is closest to a geometry. *)
	METHOD GetArcLength_ClosestTo : LREAL
	VAR_IN_OUT
		(* The geometry to check the arc length for. *)
 {attribute 'GUID' := '0554E5C0-4687-0E31-67FE-D976C958432A'}
				geometry : IPlcGeometry2D;
	END_VAR
END_METHOD

END_FUNCTION_BLOCK

// POUs/_Internal/IPlcDynamicConstraint

	{attribute 'c++_compatible'}
	{attribute 'external_name' := 'IPlcDynamicConstraint_GUID_2A75E343_6001_06F7_7543_F7E5494FC1B4'}
	{attribute 'TcIecLibraryType'}
	{attribute 'no_explicit_call' := 'do not call this POU directly'}
	{attribute 'no_assign_warning'}
	(* Internal representation of dynamic constraints. *)
	FUNCTION_BLOCK IPlcDynamicConstraint
	VAR
		{attribute 'hide'}
		_reserved0 : ULINT;
		 {attribute 'hide'}
		_reserved1 : UINT_0_32;
		 {attribute 'hide'}
		_reserved2 : ARRAY [1..4] OF UINT_8_16;
		 {attribute 'hide'}
		_reserved3 : ARRAY [1..20] OF USINT;
	END_VAR


	(* Internal method *)
	{attribute 'hide'}
	METHOD FB_init : BOOL
	VAR_INPUT
		(*  if TRUE, the retain variables are initialized (warm start / cold start) *)
		bInitRetains : BOOL;
		(*  if TRUE, the instance afterwards gets moved into the copy code (online change) *)
		bInCopyCode : BOOL;
	END_VAR
END_METHOD


	(* Internal method *)
	{attribute 'hide'}
	METHOD FB_exit : BOOL
	VAR_INPUT
		(*  if TRUE, the exit method is called for exiting an instance that is copied afterwards (online change). *)
		bInCopyCode : BOOL;
	END_VAR
END_METHOD

END_FUNCTION_BLOCK

// POUs/Dynamics/DynamicConstraint_Container

	{attribute 'c++_compatible'}
	{attribute 'external_name' := 'DynamicConstraint_Container_GUID_4E56B26A_FBB1_0E2C_6184_9B5BFD4B1F87'}
	{attribute 'TcIecLibraryType'}
	{attribute 'no_explicit_call' := 'do not call this POU directly'}
	{attribute 'no_assign_warning'}
	(* A container for dynamic constraints. *)
	FUNCTION_BLOCK DynamicConstraint_Container EXTENDS IPlcDynamicConstraint


	(* Internal method *)
	{attribute 'hide'}
	METHOD FB_init : BOOL
	VAR_INPUT
		(*  if TRUE, the retain variables are initialized (warm start / cold start) *)
		bInitRetains : BOOL;
		(*  if TRUE, the instance afterwards gets moved into the copy code (online change) *)
		bInCopyCode : BOOL;
	END_VAR
END_METHOD


	(* Internal method *)
	{attribute 'hide'}
	METHOD FB_exit : BOOL
	VAR_INPUT
		(*  if TRUE, the exit method is called for exiting an instance that is copied afterwards (online change). *)
		bInCopyCode : BOOL;
	END_VAR
END_METHOD


	(* Removes all dynamic constraints from the container. *)
	METHOD Clear
END_METHOD


	(* Adds a copy of a dynamic constraint to the container. If the dynamic constraint changes afterwards, the value in the container will not reflect that change. *)
	METHOD AddConstraint
	VAR_INPUT
		(* A reference to the constraint to be added. *)
 {attribute 'GUID' := '2A75E343-6001-06F7-7543-F7E5494FC1B4'}
				Constraint : REFERENCE TO IPlcDynamicConstraint;
	END_VAR
END_METHOD


	(* Adds a reference to a dynamic constraint to the container. If the dynamic constraint changes afterwards, the value in the container will reflect that change. *)
	METHOD AddConstraintByReference
	VAR_INPUT
		(* A reference to the constraint to be added. *)
 {attribute 'GUID' := '2A75E343-6001-06F7-7543-F7E5494FC1B4'}
				Constraint : REFERENCE TO IPlcDynamicConstraint;
	END_VAR
END_METHOD


{attribute 'monitoring' := 'call'}
	PROPERTY Count : UDINT
GET
END_GET
END_PROPERTY

END_FUNCTION_BLOCK

// POUs/Dynamics/DynamicConstraint_CartesianXY

	{attribute 'c++_compatible'}
	{attribute 'external_name' := 'DynamicConstraint_CartesianXY_GUID_03A8EDED_76EB_0EF8_4422_BD065D0A0D80'}
	{attribute 'TcIecLibraryType'}
	{attribute 'no_explicit_call' := 'do not call this POU directly'}
	(* Dynamic constraint for movement in the XY-plane, including non-tangential effects. *)
	FUNCTION_BLOCK DynamicConstraint_CartesianXY EXTENDS IPlcDynamicConstraint 
	VAR
		 {attribute 'hide'}
		_reserved1_1 : ARRAY [1..8] OF USINT;
	END_VAR


	(* Internal method *)
	{attribute 'hide'}
	METHOD FB_init : BOOL
	VAR_INPUT
		(*  if TRUE, the retain variables are initialized (warm start / cold start) *)
		bInitRetains : BOOL;
		(*  if TRUE, the instance afterwards gets moved into the copy code (online change) *)
		bInCopyCode : BOOL;
	END_VAR
END_METHOD


	(* Internal method *)
	{attribute 'hide'}
	METHOD FB_exit : BOOL
	VAR_INPUT
		(*  if TRUE, the exit method is called for exiting an instance that is copied afterwards (online change). *)
		bInCopyCode : BOOL;
	END_VAR
END_METHOD


	(* Set the dynamic limits of this instance. *)
	METHOD SetValuesVAJ
	VAR_INPUT
		(* Maximum velocity. *)
 {attribute 'GUID' := '0100FF8A-3F83-4535-990A-614CFBA4DA63'}
		 {attribute 'Namespace' := 'MC'}
				V : MC_LREAL;
		(* Maximum acceleration. *)
 {attribute 'GUID' := '0100FF8A-3F83-4535-990A-614CFBA4DA63'}
		 {attribute 'Namespace' := 'MC'}
				A : MC_LREAL;
		(* Maximum jerk. *)
 {attribute 'GUID' := '0100FF8A-3F83-4535-990A-614CFBA4DA63'}
		 {attribute 'Namespace' := 'MC'}
				J : MC_LREAL;
	END_VAR
END_METHOD


{attribute 'monitoring' := 'call'}
	PROPERTY V : MC_LREAL
GET
END_GET
SET
END_SET
END_PROPERTY


{attribute 'monitoring' := 'call'}
	PROPERTY A : MC_LREAL
GET
END_GET
SET
END_SET
END_PROPERTY


{attribute 'monitoring' := 'call'}
	PROPERTY J : MC_LREAL
GET
END_GET
SET
END_SET
END_PROPERTY

END_FUNCTION_BLOCK

// POUs/Dynamics/DynamicConstraint_CartesianXYZ

	{attribute 'c++_compatible'}
	{attribute 'external_name' := 'DynamicConstraint_CartesianXYZ_GUID_2C3E79C9_9D31_0E1B_54AF_05972CE997D0'}
	{attribute 'TcIecLibraryType'}
	{attribute 'no_explicit_call' := 'do not call this POU directly'}
	(* Dynamic constraint for movement in the XYZ-space, including non-tangential effects. *)
	FUNCTION_BLOCK DynamicConstraint_CartesianXYZ EXTENDS IPlcDynamicConstraint 
	VAR
		 {attribute 'hide'}
		_reserved1_1 : ARRAY [1..8] OF USINT;
	END_VAR


	(* Internal method *)
	{attribute 'hide'}
	METHOD FB_init : BOOL
	VAR_INPUT
		(*  if TRUE, the retain variables are initialized (warm start / cold start) *)
		bInitRetains : BOOL;
		(*  if TRUE, the instance afterwards gets moved into the copy code (online change) *)
		bInCopyCode : BOOL;
	END_VAR
END_METHOD


	(* Internal method *)
	{attribute 'hide'}
	METHOD FB_exit : BOOL
	VAR_INPUT
		(*  if TRUE, the exit method is called for exiting an instance that is copied afterwards (online change). *)
		bInCopyCode : BOOL;
	END_VAR
END_METHOD


	(* Set the dynamic limits of this instance. *)
	METHOD SetValuesVAJ
	VAR_INPUT
		(* Maximum velocity. *)
 {attribute 'GUID' := '0100FF8A-3F83-4535-990A-614CFBA4DA63'}
		 {attribute 'Namespace' := 'MC'}
				V : MC_LREAL;
		(* Maximum acceleration. *)
 {attribute 'GUID' := '0100FF8A-3F83-4535-990A-614CFBA4DA63'}
		 {attribute 'Namespace' := 'MC'}
				A : MC_LREAL;
		(* Maximum jerk. *)
 {attribute 'GUID' := '0100FF8A-3F83-4535-990A-614CFBA4DA63'}
		 {attribute 'Namespace' := 'MC'}
				J : MC_LREAL;
	END_VAR
END_METHOD


{attribute 'monitoring' := 'call'}
	PROPERTY V : MC_LREAL
GET
END_GET
SET
END_SET
END_PROPERTY


{attribute 'monitoring' := 'call'}
	PROPERTY A : MC_LREAL
GET
END_GET
SET
END_SET
END_PROPERTY


{attribute 'monitoring' := 'call'}
	PROPERTY J : MC_LREAL
GET
END_GET
SET
END_SET
END_PROPERTY

END_FUNCTION_BLOCK

// POUs/Dynamics/DynamicConstraint_Path

	{attribute 'c++_compatible'}
	{attribute 'external_name' := 'DynamicConstraint_Path_GUID_9504FC49_25E3_0E57_4820_EFCEE8D2590F'}
	{attribute 'TcIecLibraryType'}
	{attribute 'hide'}
	{attribute 'no_explicit_call' := 'do not call this POU directly'}
	{attribute 'no_assign_warning'}
	(* DEPRECATED. Please replace with either DynamicConstraint_PathXY or DynamicConstraint_Coordinates, depending on use case. *)
	FUNCTION_BLOCK DynamicConstraint_Path EXTENDS DynamicConstraint_PathXY


	(* Internal method *)
	{attribute 'hide'}
	METHOD FB_init : BOOL
	VAR_INPUT
		(*  if TRUE, the retain variables are initialized (warm start / cold start) *)
		bInitRetains : BOOL;
		(*  if TRUE, the instance afterwards gets moved into the copy code (online change) *)
		bInCopyCode : BOOL;
	END_VAR
END_METHOD


	(* Internal method *)
	{attribute 'hide'}
	METHOD FB_exit : BOOL
	VAR_INPUT
		(*  if TRUE, the exit method is called for exiting an instance that is copied afterwards (online change). *)
		bInCopyCode : BOOL;
	END_VAR
END_METHOD

END_FUNCTION_BLOCK

// POUs/Dynamics/DynamicConstraint_PathXY

	{attribute 'c++_compatible'}
	{attribute 'external_name' := 'DynamicConstraint_PathXY_GUID_8645CFB1_6915_0E93_7E4B_AF560953CDAD'}
	{attribute 'TcIecLibraryType'}
	{attribute 'no_explicit_call' := 'do not call this POU directly'}
	{attribute 'no_assign_warning'}
	(* One dimensional dynamic constraint along the XY-components of a path, ignoring non-tangential effects. *)
	FUNCTION_BLOCK DynamicConstraint_PathXY EXTENDS IPlcDynamicConstraint 
	VAR
		 {attribute 'hide'}
		_reserved1_1 : ARRAY [1..8] OF USINT;
	END_VAR


	(* Internal method *)
	{attribute 'hide'}
	METHOD FB_init : BOOL
	VAR_INPUT
		(*  if TRUE, the retain variables are initialized (warm start / cold start) *)
		bInitRetains : BOOL;
		(*  if TRUE, the instance afterwards gets moved into the copy code (online change) *)
		bInCopyCode : BOOL;
	END_VAR
END_METHOD


	(* Internal method *)
	{attribute 'hide'}
	METHOD FB_exit : BOOL
	VAR_INPUT
		(*  if TRUE, the exit method is called for exiting an instance that is copied afterwards (online change). *)
		bInCopyCode : BOOL;
	END_VAR
END_METHOD


	(* Set the dynamic limits of this instance. *)
	METHOD SetValuesVADJ
	VAR_INPUT
		(* Maximum velocity. *)
 {attribute 'GUID' := '0100FF8A-3F83-4535-990A-614CFBA4DA63'}
		 {attribute 'Namespace' := 'MC'}
				V : MC_LREAL;
		(* Maximum acceleration. *)
 {attribute 'GUID' := '0100FF8A-3F83-4535-990A-614CFBA4DA63'}
		 {attribute 'Namespace' := 'MC'}
				A : MC_LREAL;
		(* Maximum deceleration. *)
 {attribute 'GUID' := '0100FF8A-3F83-4535-990A-614CFBA4DA63'}
		 {attribute 'Namespace' := 'MC'}
				D : MC_LREAL;
		(* Maximum jerk. *)
 {attribute 'GUID' := '0100FF8A-3F83-4535-990A-614CFBA4DA63'}
		 {attribute 'Namespace' := 'MC'}
				J : MC_LREAL;
	END_VAR
END_METHOD


{attribute 'monitoring' := 'call'}
	PROPERTY V : MC_LREAL
GET
END_GET
SET
END_SET
END_PROPERTY


{attribute 'monitoring' := 'call'}
	PROPERTY A : MC_LREAL
GET
END_GET
SET
END_SET
END_PROPERTY


{attribute 'monitoring' := 'call'}
	PROPERTY D : MC_LREAL
GET
END_GET
SET
END_SET
END_PROPERTY


{attribute 'monitoring' := 'call'}
	PROPERTY J : MC_LREAL
GET
END_GET
SET
END_SET
END_PROPERTY

END_FUNCTION_BLOCK

// POUs/Dynamics/DynamicConstraint_Coordinates

	{attribute 'c++_compatible'}
	{attribute 'external_name' := 'DynamicConstraint_Coordinates_GUID_C1835B09_32E2_02A7_6737_49CAC3594837'}
	{attribute 'TcIecLibraryType'}
	{attribute 'no_explicit_call' := 'do not call this POU directly'}
	{attribute 'no_assign_warning'}
	(* Dynamic constraints for individual coordinates. *)
	FUNCTION_BLOCK DynamicConstraint_Coordinates EXTENDS IPlcDynamicConstraint


	(* Internal method *)
	{attribute 'hide'}
	METHOD FB_init : BOOL
	VAR_INPUT
		(*  if TRUE, the retain variables are initialized (warm start / cold start) *)
		bInitRetains : BOOL;
		(*  if TRUE, the instance afterwards gets moved into the copy code (online change) *)
		bInCopyCode : BOOL;
	END_VAR
END_METHOD


	(* Internal method *)
	{attribute 'hide'}
	METHOD FB_exit : BOOL
	VAR_INPUT
		(*  if TRUE, the exit method is called for exiting an instance that is copied afterwards (online change). *)
		bInCopyCode : BOOL;
	END_VAR
END_METHOD


	(* Adds limits for a specific coordinate. If the coordinate is already limited, limits are merged. *)
	METHOD AddLimit
	VAR_INPUT
		(* Coordinate type. E.g. Coord_Mcs_X, Coord_Mcs_Y, ... *)
 {attribute 'GUID' := 'ABF37E9D-1614-4226-99CD-162368D15A32'}
				Coordinate : CoordinateType;
		(* Maximum velocity. *)
 {attribute 'GUID' := '0100FF8A-3F83-4535-990A-614CFBA4DA63'}
		 {attribute 'Namespace' := 'MC'}
				V : MC_LREAL;
		(* Maximum acceleration. *)
 {attribute 'GUID' := '0100FF8A-3F83-4535-990A-614CFBA4DA63'}
		 {attribute 'Namespace' := 'MC'}
				A : MC_LREAL;
		(* Maximum deceleration. *)
 {attribute 'GUID' := '0100FF8A-3F83-4535-990A-614CFBA4DA63'}
		 {attribute 'Namespace' := 'MC'}
				D : MC_LREAL;
		(* Maximum jerk. *)
 {attribute 'GUID' := '0100FF8A-3F83-4535-990A-614CFBA4DA63'}
		 {attribute 'Namespace' := 'MC'}
				J : MC_LREAL;
	END_VAR
END_METHOD


	(* Sets limits for a specific coordinate. If the coordinate is already limited, existing limits are overwritten. *)
	METHOD SetLimit
	VAR_INPUT
		(* Coordinate type. E.g. Coord_Mcs_X, Coord_Mcs_Y, ... *)
 {attribute 'GUID' := 'ABF37E9D-1614-4226-99CD-162368D15A32'}
				Coordinate : CoordinateType;
		(* Maximum velocity. *)
 {attribute 'GUID' := '0100FF8A-3F83-4535-990A-614CFBA4DA63'}
		 {attribute 'Namespace' := 'MC'}
				V : MC_LREAL;
		(* Maximum acceleration. *)
 {attribute 'GUID' := '0100FF8A-3F83-4535-990A-614CFBA4DA63'}
		 {attribute 'Namespace' := 'MC'}
				A : MC_LREAL;
		(* Maximum deceleration. *)
 {attribute 'GUID' := '0100FF8A-3F83-4535-990A-614CFBA4DA63'}
		 {attribute 'Namespace' := 'MC'}
				D : MC_LREAL;
		(* Maximum jerk. *)
 {attribute 'GUID' := '0100FF8A-3F83-4535-990A-614CFBA4DA63'}
		 {attribute 'Namespace' := 'MC'}
				J : MC_LREAL;
	END_VAR
END_METHOD


	(* Removes limits for a specific coordinate. *)
	METHOD RemoveLimit
	VAR_INPUT
		(* Coordinate type. E.g. Coord_Mcs_X, Coord_Mcs_Y, ... *)
 {attribute 'GUID' := 'ABF37E9D-1614-4226-99CD-162368D15A32'}
				Coordinate : CoordinateType;
	END_VAR
END_METHOD


	(* Removes limits for all coordinates. *)
	METHOD Clear
END_METHOD


	(* Gets the contained velocity limit for a specific coordinate. If no limits for the coordinate are set, returns MC_INVALID. *)
	METHOD GetV : MC_LREAL
	VAR_INPUT
		(* Coordinate type. E.g. Coord_Mcs_X, Coord_Mcs_Y, ... *)
 {attribute 'GUID' := 'ABF37E9D-1614-4226-99CD-162368D15A32'}
				Coordinate : CoordinateType;
	END_VAR
END_METHOD


	(* Gets the contained acceleration limit for a specific coordinate. If no limits for the coordinate are set, returns MC_INVALID. *)
	METHOD GetA : MC_LREAL
	VAR_INPUT
		(* Coordinate type. E.g. Coord_Mcs_X, Coord_Mcs_Y, ... *)
 {attribute 'GUID' := 'ABF37E9D-1614-4226-99CD-162368D15A32'}
				Coordinate : CoordinateType;
	END_VAR
END_METHOD


	(* Gets the contained deceleration limit for a specific coordinate. If no limits for the coordinate are set, returns MC_INVALID. *)
	METHOD GetD : MC_LREAL
	VAR_INPUT
		(* Coordinate type. E.g. Coord_Mcs_X, Coord_Mcs_Y, ... *)
 {attribute 'GUID' := 'ABF37E9D-1614-4226-99CD-162368D15A32'}
				Coordinate : CoordinateType;
	END_VAR
END_METHOD


	(* Gets the contained jerk limit for a specific coordinate. If no limits for the coordinate are set, returns MC_INVALID. *)
	METHOD GetJ : MC_LREAL
	VAR_INPUT
		(* Coordinate type. E.g. Coord_Mcs_X, Coord_Mcs_Y, ... *)
 {attribute 'GUID' := 'ABF37E9D-1614-4226-99CD-162368D15A32'}
				Coordinate : CoordinateType;
	END_VAR
END_METHOD


{attribute 'monitoring' := 'call'}
	PROPERTY Count : UDINT
GET
END_GET
END_PROPERTY

END_FUNCTION_BLOCK

// POUs/Dynamics/DynamicConstraint_PathXYZ

	{attribute 'c++_compatible'}
	{attribute 'external_name' := 'DynamicConstraint_PathXYZ_GUID_D3A3B83F_025A_025E_473F_7BB1D6E7E254'}
	{attribute 'TcIecLibraryType'}
	{attribute 'no_explicit_call' := 'do not call this POU directly'}
	(* One dimensional dynamic constraint along the XYZ-components of a path, ignoring non-tangential effects. *)
	FUNCTION_BLOCK DynamicConstraint_PathXYZ EXTENDS IPlcDynamicConstraint 
	VAR
		 {attribute 'hide'}
		_reserved1_1 : ARRAY [1..8] OF USINT;
	END_VAR


	(* Internal method *)
	{attribute 'hide'}
	METHOD FB_init : BOOL
	VAR_INPUT
		(*  if TRUE, the retain variables are initialized (warm start / cold start) *)
		bInitRetains : BOOL;
		(*  if TRUE, the instance afterwards gets moved into the copy code (online change) *)
		bInCopyCode : BOOL;
	END_VAR
END_METHOD


	(* Internal method *)
	{attribute 'hide'}
	METHOD FB_exit : BOOL
	VAR_INPUT
		(*  if TRUE, the exit method is called for exiting an instance that is copied afterwards (online change). *)
		bInCopyCode : BOOL;
	END_VAR
END_METHOD


	(* Set the dynamic limits of this instance. *)
	METHOD SetValuesVADJ
	VAR_INPUT
		(* Maximum velocity. *)
 {attribute 'GUID' := '0100FF8A-3F83-4535-990A-614CFBA4DA63'}
		 {attribute 'Namespace' := 'MC'}
				V : MC_LREAL;
		(* Maximum acceleration. *)
 {attribute 'GUID' := '0100FF8A-3F83-4535-990A-614CFBA4DA63'}
		 {attribute 'Namespace' := 'MC'}
				A : MC_LREAL;
		(* Maximum deceleration. *)
 {attribute 'GUID' := '0100FF8A-3F83-4535-990A-614CFBA4DA63'}
		 {attribute 'Namespace' := 'MC'}
				D : MC_LREAL;
		(* Maximum jerk. *)
 {attribute 'GUID' := '0100FF8A-3F83-4535-990A-614CFBA4DA63'}
		 {attribute 'Namespace' := 'MC'}
				J : MC_LREAL;
	END_VAR
END_METHOD


{attribute 'monitoring' := 'call'}
	PROPERTY V : MC_LREAL
GET
END_GET
SET
END_SET
END_PROPERTY


{attribute 'monitoring' := 'call'}
	PROPERTY A : MC_LREAL
GET
END_GET
SET
END_SET
END_PROPERTY


{attribute 'monitoring' := 'call'}
	PROPERTY D : MC_LREAL
GET
END_GET
SET
END_SET
END_PROPERTY


{attribute 'monitoring' := 'call'}
	PROPERTY J : MC_LREAL
GET
END_GET
SET
END_SET
END_PROPERTY

END_FUNCTION_BLOCK

// POUs/Dynamics/DynamicProfile_7phase

	{attribute 'c++_compatible'}
	{attribute 'external_name' := 'DynamicProfile_7phase_GUID_BBFEA9C1_675A_0BDC_5499_6C1D63BB7AA5'}
	{attribute 'TcIecLibraryType'}
	{attribute 'no_explicit_call' := 'do not call this POU directly'}
	{attribute 'no_assign'}
	(* Calculate a dynamic profile with up to seven phases between start and end point in some dynamic limits. *)
	FUNCTION_BLOCK DynamicProfile_7phase
	VAR
		(* Maximum (=-minimum) velocity. *)
		maximumVelocity : LREAL;
		(* Maximum (=-minimum) acceleration. *)
		maximumAcceleration : LREAL;
		(* Maximum (=-minimum) jerk. *)
		maximumJerk : LREAL;
	END_VAR
	VAR_OUTPUT
		(* is the profile valid? *)
		validProfile : BOOL;
	END_VAR
	VAR
		 {attribute 'hide'}
		_reserved1 : UINT_24_56;
		 {attribute 'hide'}
		_reserved2 : ARRAY [1..4] OF UINT_8_16;
		 {attribute 'hide'}
		_reserved3 : ARRAY [1..8] OF USINT;
	END_VAR


	(* Internal method *)
	{attribute 'hide'}
	METHOD FB_init : BOOL
	VAR_INPUT
		(*  if TRUE, the retain variables are initialized (warm start / cold start) *)
		bInitRetains : BOOL;
		(*  if TRUE, the instance afterwards gets moved into the copy code (online change) *)
		bInCopyCode : BOOL;
	END_VAR
END_METHOD


	(* Internal method *)
	{attribute 'hide'}
	METHOD FB_exit : BOOL
	VAR_INPUT
		(*  if TRUE, the exit method is called for exiting an instance that is copied afterwards (online change). *)
		bInCopyCode : BOOL;
	END_VAR
END_METHOD


	(* Set the dynamic limits for the profile. *)
	METHOD SetDynamicLimits
	VAR_INPUT
		(* Maximum (=-minimum) velocity of the profile. *)
		maximumVelocity : LREAL;
		(* Maximum (=-minimum) acceleration of the profile. *)
		maximumAcceleration : LREAL;
		(* Maximum (=-minimum) jerk of the profile. *)
		maximumJerk : LREAL;
	END_VAR
END_METHOD


	(* Calculates the dynamic profile from initial to final distance. *)
	METHOD CalculateProfile
	VAR_INPUT
		(* Inital distance (position) of the profile. *)
		initialDistance : LREAL;
		(* Inital velocity of the profile. *)
		initialVelocity : LREAL;
		(* Inital acceleration of the profile. *)
		initialAcceleration : LREAL;
		(* Final distance (position) of the profile. *)
		finalDistance : LREAL;
		(* Final velocity of the profile. *)
		finalVelocity : LREAL;
		(* Final acceleration of the profile. *)
		finalAcceleration : LREAL;
	END_VAR
END_METHOD


	(* Evaluates the profile at given time within this profile. *)
	METHOD GetValues
	VAR_INPUT
		(* Time within this profile where the dynamic profile is evaluated. *)
		_time : LREAL;
	END_VAR
	VAR_IN_OUT
		(* Distance (position). *)
		distance : LREAL;
		(* Velocity. *)
		velocity : LREAL;
		(* Acceleration. *)
		acceleration : LREAL;
	END_VAR
END_METHOD


	(* Returns the total time needed for this dynamic profile. *)
	METHOD GetDuration : LREAL
END_METHOD

END_FUNCTION_BLOCK

// POUs/Dynamics/DynamicProfile_3phase

	{attribute 'c++_compatible'}
	{attribute 'external_name' := 'DynamicProfile_3phase_GUID_D0BCE02C_50FC_0D8E_7F1F_AC94CB11E780'}
	{attribute 'TcIecLibraryType'}
	{attribute 'no_explicit_call' := 'do not call this POU directly'}
	{attribute 'no_assign'}
	(* Calculate a dynamic profile with up to three phases between start and end point in some dynamic limits. *)
	FUNCTION_BLOCK DynamicProfile_3phase
	VAR
		(* Maximum (=-minimum) velocity. *)
		maximumVelocity : LREAL;
		(* Maximum (=-minimum) acceleration. *)
		maximumAcceleration : LREAL;
		(* Maximum (=-minimum) jerk. *)
		maximumJerk : LREAL;
	END_VAR
	VAR_OUTPUT
		(* is the profile valid? *)
		validProfile : BOOL;
	END_VAR
	VAR
		 {attribute 'hide'}
		_reserved1 : UINT_24_56;
		 {attribute 'hide'}
		_reserved2 : ARRAY [1..4] OF UINT_8_16;
		 {attribute 'hide'}
		_reserved3 : ARRAY [1..8] OF USINT;
	END_VAR


	(* Internal method *)
	{attribute 'hide'}
	METHOD FB_init : BOOL
	VAR_INPUT
		(*  if TRUE, the retain variables are initialized (warm start / cold start) *)
		bInitRetains : BOOL;
		(*  if TRUE, the instance afterwards gets moved into the copy code (online change) *)
		bInCopyCode : BOOL;
	END_VAR
END_METHOD


	(* Internal method *)
	{attribute 'hide'}
	METHOD FB_exit : BOOL
	VAR_INPUT
		(*  if TRUE, the exit method is called for exiting an instance that is copied afterwards (online change). *)
		bInCopyCode : BOOL;
	END_VAR
END_METHOD


	(* Set the dynamic limits for the profile. *)
	METHOD SetDynamicLimits
	VAR_INPUT
		(* Maximum (=-minimum) velocity of the profile. *)
		maximumVelocity : LREAL;
		(* Maximum (=-minimum) acceleration of the profile. *)
		maximumAcceleration : LREAL;
		(* Maximum (=-minimum) jerk of the profile. *)
		maximumJerk : LREAL;
	END_VAR
END_METHOD


	(* Calculates the dynamic profile from initial to final distance. *)
	METHOD CalculateProfile
	VAR_INPUT
		(* Inital distance (position) of the profile. *)
		initialDistance : LREAL;
		(* Inital velocity of the profile. *)
		initialVelocity : LREAL;
		(* Inital acceleration of the profile. *)
		initialAcceleration : LREAL;
		(* Final velocity of the profile. *)
		finalVelocity : LREAL;
		(* Final acceleration of the profile. *)
		finalAcceleration : LREAL;
	END_VAR
END_METHOD


	(* Evaluates the profile at given time within this profile. *)
	METHOD GetValues
	VAR_INPUT
		(* Time within this profile where the dynamic profile is evaluated. *)
		_time : LREAL;
	END_VAR
	VAR_IN_OUT
		(* Distance (position). *)
		distance : LREAL;
		(* Velocity. *)
		velocity : LREAL;
		(* Acceleration. *)
		acceleration : LREAL;
	END_VAR
END_METHOD


	(* Returns the total time needed for this dynamic profile. *)
	METHOD GetDuration : LREAL
END_METHOD

END_FUNCTION_BLOCK

// POUs/Coordinates/GetMcsCoordinateType

	{attribute 'TcIecLibraryType'}
	{attribute 'external_name' := 'GetMcsCoordinateType_GUID_70E22AD0_D1F9_09B3_6577_642E30639DFB'}
	(* Creates a CoordinateType FB from E_McsCoordType. *)
	FUNCTION GetMcsCoordinateType : CoordinateType
	VAR_INPUT
		mcsType	:	E_McsCoordType;	(* Mcs coordinate type. *)
	END_VAR

END_FUNCTION

// POUs/Coordinates/GetUninterpretedCoordinateType

	{attribute 'TcIecLibraryType'}
	{attribute 'external_name' := 'GetUninterpretedCoordinateType_GUID_78519344_AE40_0BCA_4E46_ED752C25D558'}
	(* Creates a CoordinateType FB from an index. *)
	FUNCTION GetUninterpretedCoordinateType : CoordinateType
	VAR_INPUT
		mcsType	:	UDINT;	(* Mcs coordinate type. *)
	END_VAR

END_FUNCTION

// POUs/Spatial/Functions/ConcatenateXY

	{attribute 'TcIecLibraryType'}
	{attribute 'external_name' := 'ConcatenateXY_GUID_EE46346B_E4F7_0BD3_4A74_B568C54FDC42'}
	(* Concatenate two instances of PositionXY. *)
	FUNCTION ConcatenateXY : BOOL
	VAR_IN_OUT
		position0	:	PositionXY;	(* 1st input position of the concatenation. *)
		position1	:	PositionXY;	(* 2nd input position of the concatenation. *)
		concatenation	:	PositionXY;	(* The concatenation of the two input instances. *)
	END_VAR

END_FUNCTION

// POUs/Spatial/Functions/Concatenate3D

	{attribute 'TcIecLibraryType'}
	{attribute 'external_name' := 'Concatenate3D_GUID_8E8FF55D_CB0F_02DD_65DD_FC333C596E8C'}
	(* Concatenate two instances of Position3D. *)
	FUNCTION Concatenate3D : BOOL
	VAR_IN_OUT
		position0	:	Position3D;	(* 1st input position of the concatenation. *)
		position1	:	Position3D;	(* 2nd input position of the concatenation. *)
		concatenation	:	Position3D;	(* The concatenation of the two input instances. *)
	END_VAR

END_FUNCTION

// POUs/Spatial/Functions/ConcatenateC

	{attribute 'TcIecLibraryType'}
	{attribute 'external_name' := 'ConcatenateC_GUID_E4B3CD11_B18A_01BE_7BAF_D2E3F242089F'}
	(* Concatenate two instances Orientation2D. *)
	FUNCTION ConcatenateC : BOOL
	VAR_IN_OUT
		rotation0	:	Orientation2D;	(* 1st input orientation of the concatenation. *)
		rotation1	:	Orientation2D;	(* 2nd input orientation of the concatenation. *)
		concatenation	:	Orientation2D;	(* The concatenation of the two input instances. *)
	END_VAR

END_FUNCTION

// POUs/Spatial/Positions/Orientation2D

	{attribute 'c++_compatible'}
	{attribute 'external_name' := 'Orientation2D_GUID_ABCF5F54_5133_060C_4FEE_702387088411'}
	{attribute 'TcIecLibraryType'}
	{attribute 'no_explicit_call' :='do not call this POU directly'}
	{attribute 'no_assign'}
	(* 2D orientation. Angle in degrees [Â°]. *)
	FUNCTION_BLOCK Orientation2D
	VAR
		(* Rotation angle in degrees [Â°]. *)
		phi : LREAL;
		 {attribute 'hide'}
		_reserved1 : ARRAY [1..80] OF USINT;
	END_VAR


